Yaskawa INFORM job: A_ROOF_SIDE_0617_2_PAINT_30.JBI

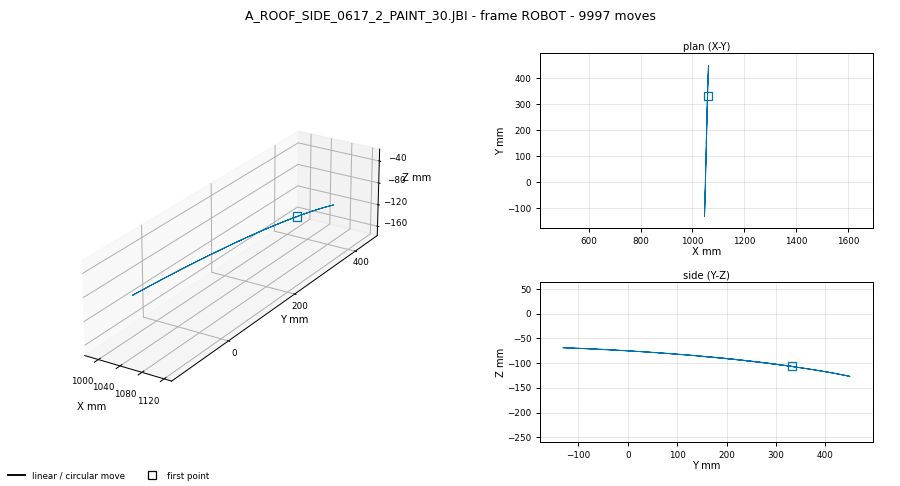
[picture p0: tool path of A_ROOF_SIDE_0617_2_PAINT_30.JBI in frame ROBOT, 9997 of 9997 moves have a stored position in this frame; points joined in program order, loops and branches not executed]
/JOB
//NAME A_ROOF_SIDE_0617_2_PAINT30
//POS
///NPOS 9997,0,0,0,0,0
///TOOL 1
///USER 0
///POSTYPE ROBOT
///RECTAN
///RCONF 1,0,0,0,0,0,0,0,0,0,0,0,0,0,0,0,0,0,0,0,0,0,0,0
C00000=1058.571,332.665,-106.204,173.587,36.326,156.830
C00001=1058.564,332.417,-106.170,173.583,36.321,156.829
C00002=1058.557,332.167,-106.134,173.579,36.317,156.828
C00003=1058.551,331.916,-106.099,173.576,36.312,156.827
C00004=1058.545,331.666,-106.063,173.572,36.307,156.826
C00005=1058.538,331.416,-106.028,173.567,36.303,156.825
C00006=1058.532,331.169,-105.993,173.564,36.298,156.824
C00007=1058.525,330.921,-105.958,173.560,36.294,156.823
C00008=1058.518,330.674,-105.923,173.557,36.289,156.822
C00009=1058.512,330.426,-105.889,173.553,36.285,156.821
C00010=1058.504,330.179,-105.854,173.548,36.280,156.820
C00011=1058.498,329.932,-105.819,173.545,36.276,156.819
C00012=1058.491,329.684,-105.785,173.541,36.271,156.818
C00013=1058.484,329.436,-105.750,173.538,36.267,156.817
C00014=1058.477,329.189,-105.716,173.534,36.262,156.816
C00015=1058.471,328.941,-105.681,173.530,36.258,156.815
C00016=1058.464,328.693,-105.646,173.526,36.254,156.814
C00017=1058.457,328.446,-105.612,173.523,36.249,156.813
C00018=1058.451,328.199,-105.578,173.519,36.245,156.812
C00019=1058.444,327.951,-105.543,173.516,36.241,156.811
C00020=1058.437,327.704,-105.509,173.511,36.237,156.810
C00021=1058.430,327.456,-105.474,173.507,36.232,156.809
C00022=1058.423,327.208,-105.440,173.504,36.227,156.808
C00023=1058.416,326.961,-105.405,173.500,36.223,156.807
C00024=1058.410,326.713,-105.371,173.497,36.219,156.806
C00025=1058.403,326.466,-105.337,173.493,36.215,156.805
C00026=1058.396,326.219,-105.302,173.490,36.210,156.804
C00027=1058.390,325.971,-105.268,173.485,36.206,156.803
C00028=1058.383,325.723,-105.234,173.482,36.202,156.802
C00029=1058.376,325.475,-105.200,173.478,36.197,156.801
C00030=1058.370,325.228,-105.165,173.475,36.193,156.801
C00031=1058.363,324.981,-105.131,173.471,36.189,156.800
C00032=1058.356,324.733,-105.097,173.468,36.184,156.799
C00033=1058.349,324.485,-105.063,173.464,36.180,156.798
C00034=1058.343,324.238,-105.029,173.461,36.176,156.797
C00035=1058.337,323.990,-104.994,173.456,36.171,156.796
C00036=1058.329,323.743,-104.960,173.453,36.167,156.795
C00037=1058.324,323.495,-104.926,173.449,36.163,156.794
C00038=1058.316,323.248,-104.892,173.446,36.159,156.793
C00039=1058.310,323.000,-104.857,173.442,36.154,156.792
C00040=1058.303,322.753,-104.824,173.438,36.150,156.791
C00041=1058.297,322.505,-104.790,173.435,36.145,156.790
C00042=1058.290,322.257,-104.755,173.431,36.141,156.789
C00043=1058.284,322.010,-104.722,173.428,36.137,156.788
C00044=1058.277,321.762,-104.687,173.424,36.133,156.787
C00045=1058.270,321.514,-104.653,173.421,36.128,156.786
C00046=1058.264,321.267,-104.619,173.417,36.124,156.785
C00047=1058.257,321.019,-104.586,173.414,36.120,156.784
C00048=1058.251,320.772,-104.551,173.410,36.116,156.783
C00049=1058.245,320.524,-104.517,173.407,36.112,156.783
C00050=1058.238,320.276,-104.484,173.403,36.107,156.781
C00051=1058.232,320.028,-104.450,173.399,36.103,156.781
C00052=1058.225,319.781,-104.416,173.395,36.099,156.780
C00053=1058.219,319.533,-104.382,173.392,36.094,156.779
C00054=1058.212,319.286,-104.348,173.388,36.090,156.778
C00055=1058.206,319.038,-104.314,173.385,36.086,156.777
C00056=1058.199,318.791,-104.280,173.381,36.082,156.776
C00057=1058.193,318.543,-104.247,173.378,36.078,156.775
C00058=1058.186,318.287,-104.212,173.374,36.073,156.774
C00059=1058.179,318.031,-104.177,173.371,36.069,156.773
C00060=1058.173,317.776,-104.143,173.367,36.064,156.772
C00061=1058.166,317.521,-104.107,173.364,36.060,156.771
C00062=1058.160,317.273,-104.074,173.360,36.056,156.770
C00063=1058.153,317.025,-104.040,173.357,36.052,156.769
C00064=1058.147,316.778,-104.006,173.353,36.047,156.768
C00065=1058.141,316.529,-103.973,173.350,36.043,156.767
C00066=1058.134,316.282,-103.939,173.346,36.039,156.767
C00067=1058.128,316.035,-103.905,173.343,36.034,156.766
C00068=1058.121,315.787,-103.872,173.339,36.030,156.765
C00069=1058.115,315.540,-103.838,173.336,36.026,156.764
C00070=1058.108,315.291,-103.805,173.333,36.022,156.763
C00071=1058.103,315.044,-103.771,173.329,36.018,156.762
C00072=1058.096,314.796,-103.738,173.326,36.014,156.761
C00073=1058.090,314.548,-103.704,173.323,36.010,156.760
C00074=1058.084,314.301,-103.671,173.320,36.006,156.759
C00075=1058.078,314.054,-103.637,173.316,36.001,156.758
C00076=1058.071,313.805,-103.604,173.313,35.997,156.757
C00077=1058.064,313.558,-103.570,173.309,35.993,156.756
C00078=1058.058,313.311,-103.538,173.306,35.989,156.756
C00079=1058.051,313.063,-103.504,173.302,35.985,156.755
C00080=1058.044,312.815,-103.471,173.299,35.981,156.754
C00081=1058.038,312.567,-103.438,173.295,35.977,156.753
C00082=1058.031,312.320,-103.405,173.292,35.973,156.752
C00083=1058.025,312.073,-103.372,173.288,35.969,156.751
C00084=1058.018,311.824,-103.339,173.285,35.964,156.750
C00085=1058.011,311.577,-103.306,173.282,35.960,156.749
C00086=1058.005,311.328,-103.273,173.278,35.956,156.748
C00087=1057.998,311.081,-103.239,173.275,35.952,156.748
C00088=1057.992,310.834,-103.207,173.271,35.948,156.747
C00089=1057.985,310.586,-103.174,173.268,35.944,156.746
C00090=1057.978,310.338,-103.141,173.264,35.940,156.745
C00091=1057.972,310.090,-103.108,173.262,35.937,156.744
C00092=1057.965,309.843,-103.074,173.258,35.933,156.743
C00093=1057.958,309.595,-103.042,173.255,35.929,156.742
C00094=1057.952,309.348,-103.009,173.252,35.924,156.742
C00095=1057.945,309.100,-102.977,173.248,35.920,156.741
C00096=1057.938,308.852,-102.943,173.245,35.916,156.740
C00097=1057.932,308.604,-102.911,173.241,35.912,156.739
C00098=1057.926,308.357,-102.878,173.238,35.908,156.738
C00099=1057.920,308.109,-102.845,173.234,35.904,156.737
C00100=1057.913,307.861,-102.812,173.231,35.901,156.736
C00101=1057.906,307.613,-102.779,173.228,35.897,156.736
C00102=1057.900,307.366,-102.747,173.225,35.893,156.735
C00103=1057.893,307.118,-102.714,173.222,35.888,156.734
C00104=1057.886,306.870,-102.681,173.218,35.884,156.733
C00105=1057.880,306.622,-102.649,173.215,35.880,156.732
C00106=1057.874,306.375,-102.616,173.211,35.876,156.731
C00107=1057.867,306.127,-102.583,173.208,35.873,156.730
C00108=1057.861,305.880,-102.550,173.204,35.869,156.730
C00109=1057.855,305.632,-102.518,173.202,35.865,156.729
C00110=1057.847,305.384,-102.486,173.199,35.861,156.728
C00111=1057.841,305.136,-102.453,173.195,35.857,156.727
C00112=1057.835,304.888,-102.420,173.192,35.852,156.726
C00113=1057.829,304.641,-102.388,173.188,35.849,156.725
C00114=1057.822,304.389,-102.355,173.185,35.845,156.724
C00115=1057.816,304.138,-102.321,173.182,35.841,156.724
C00116=1057.809,303.886,-102.289,173.179,35.837,156.723
C00117=1057.803,303.635,-102.256,173.176,35.833,156.722
C00118=1057.796,303.387,-102.223,173.172,35.829,156.721
C00119=1057.790,303.139,-102.190,173.169,35.825,156.720
C00120=1057.784,302.891,-102.158,173.165,35.820,156.719
C00121=1057.777,302.644,-102.126,173.163,35.817,156.718
C00122=1057.771,302.396,-102.093,173.160,35.813,156.718
C00123=1057.765,302.148,-102.061,173.156,35.809,156.717
C00124=1057.758,301.901,-102.029,173.153,35.805,156.716
C00125=1057.752,301.653,-101.996,173.149,35.801,156.715
C00126=1057.745,301.404,-101.964,173.147,35.797,156.714
C00127=1057.739,301.157,-101.931,173.143,35.793,156.713
C00128=1057.733,300.909,-101.900,173.140,35.789,156.712
C00129=1057.727,300.662,-101.867,173.137,35.785,156.712
C00130=1057.721,300.414,-101.834,173.134,35.781,156.711
C00131=1057.714,300.166,-101.803,173.131,35.777,156.710
C00132=1057.708,299.919,-101.770,173.127,35.773,156.709
C00133=1057.702,299.670,-101.738,173.124,35.769,156.708
C00134=1057.695,299.423,-101.705,173.122,35.766,156.707
C00135=1057.689,299.175,-101.673,173.118,35.762,156.707
C00136=1057.682,298.927,-101.641,173.115,35.757,156.706
C00137=1057.676,298.679,-101.609,173.111,35.753,156.705
C00138=1057.670,298.431,-101.576,173.109,35.750,156.704
C00139=1057.664,298.183,-101.544,173.106,35.746,156.703
C00140=1057.657,297.935,-101.513,173.102,35.742,156.702
C00141=1057.651,297.688,-101.480,173.099,35.738,156.701
C00142=1057.645,297.440,-101.448,173.096,35.734,156.701
C00143=1057.640,297.192,-101.416,173.093,35.730,156.700
C00144=1057.633,296.945,-101.384,173.090,35.726,156.699
C00145=1057.627,296.697,-101.352,173.087,35.722,156.698
C00146=1057.621,296.448,-101.320,173.084,35.718,156.697
C00147=1057.614,296.201,-101.288,173.080,35.714,156.696
C00148=1057.608,295.953,-101.256,173.077,35.711,156.696
C00149=1057.601,295.705,-101.225,173.075,35.707,156.695
C00150=1057.594,295.457,-101.193,173.071,35.703,156.694
C00151=1057.588,295.209,-101.160,173.068,35.699,156.693
C00152=1057.582,294.962,-101.129,173.065,35.695,156.692
C00153=1057.576,294.714,-101.097,173.062,35.691,156.692
C00154=1057.569,294.466,-101.066,173.059,35.687,156.691
C00155=1057.563,294.218,-101.034,173.055,35.684,156.690
C00156=1057.556,293.970,-101.002,173.053,35.680,156.689
C00157=1057.550,293.722,-100.971,173.050,35.676,156.688
C00158=1057.544,293.474,-100.939,173.046,35.672,156.688
C00159=1057.537,293.226,-100.907,173.044,35.669,156.687
C00160=1057.530,292.979,-100.876,173.040,35.664,156.686
C00161=1057.524,292.731,-100.844,173.037,35.661,156.685
C00162=1057.518,292.483,-100.812,173.035,35.657,156.684
C00163=1057.511,292.235,-100.781,173.031,35.653,156.684
C00164=1057.505,291.987,-100.749,173.028,35.649,156.683
C00165=1057.498,291.739,-100.717,173.026,35.646,156.682
C00166=1057.492,291.497,-100.687,173.022,35.642,156.681
C00167=1057.486,291.256,-100.656,173.019,35.638,156.680
C00168=1057.480,291.014,-100.626,173.016,35.635,156.680
C00169=1057.474,290.772,-100.595,173.013,35.630,156.679
C00170=1057.468,290.530,-100.564,173.011,35.627,156.678
C00171=1057.462,290.287,-100.533,173.007,35.623,156.677
C00172=1057.456,290.045,-100.503,173.005,35.620,156.676
C00173=1057.449,289.804,-100.472,173.002,35.616,156.676
C00174=1057.443,289.556,-100.441,172.998,35.612,156.675
C00175=1057.437,289.308,-100.409,172.996,35.608,156.674
C00176=1057.430,289.061,-100.378,172.993,35.605,156.673
C00177=1057.424,288.812,-100.347,172.989,35.601,156.673
C00178=1057.418,288.565,-100.316,172.987,35.597,156.672
C00179=1057.411,288.317,-100.284,172.983,35.593,156.671
C00180=1057.405,288.069,-100.253,172.981,35.589,156.670
C00181=1057.398,287.820,-100.222,172.978,35.586,156.669
C00182=1057.392,287.573,-100.191,172.974,35.582,156.669
C00183=1057.385,287.325,-100.160,172.972,35.578,156.668
C00184=1057.379,287.077,-100.129,172.969,35.575,156.667
C00185=1057.372,286.829,-100.097,172.966,35.571,156.666
C00186=1057.366,286.581,-100.066,172.963,35.567,156.665
C00187=1057.360,286.333,-100.035,172.960,35.563,156.665
C00188=1057.354,286.085,-100.004,172.957,35.560,156.664
C00189=1057.347,285.837,-99.972,172.954,35.556,156.663
C00190=1057.341,285.589,-99.942,172.952,35.552,156.662
C00191=1057.334,285.341,-99.910,172.948,35.549,156.662
C00192=1057.328,285.093,-99.880,172.945,35.545,156.661
C00193=1057.322,284.845,-99.849,172.943,35.541,156.660
C00194=1057.315,284.597,-99.818,172.939,35.538,156.659
C00195=1057.309,284.349,-99.786,172.937,35.533,156.658
C00196=1057.303,284.101,-99.756,172.933,35.530,156.658
C00197=1057.296,283.853,-99.725,172.930,35.526,156.657
C00198=1057.290,283.605,-99.694,172.928,35.522,156.656
C00199=1057.284,283.358,-99.663,172.924,35.519,156.655
C00200=1057.277,283.109,-99.632,172.922,35.515,156.655
C00201=1057.271,282.861,-99.602,172.919,35.511,156.654
C00202=1057.265,282.613,-99.570,172.916,35.508,156.653
C00203=1057.259,282.365,-99.540,172.913,35.504,156.652
C00204=1057.252,282.118,-99.509,172.911,35.500,156.651
C00205=1057.246,281.869,-99.478,172.907,35.496,156.651
C00206=1057.240,281.621,-99.448,172.905,35.493,156.650
C00207=1057.233,281.373,-99.416,172.902,35.489,156.649
C00208=1057.227,281.125,-99.386,172.898,35.485,156.648
C00209=1057.221,280.877,-99.355,172.896,35.482,156.648
C00210=1057.215,280.630,-99.324,172.893,35.477,156.647
C00211=1057.208,280.381,-99.293,172.890,35.474,156.646
C00212=1057.203,280.133,-99.263,172.887,35.470,156.645
C00213=1057.196,279.885,-99.232,172.885,35.466,156.644
C00214=1057.189,279.637,-99.201,172.881,35.463,156.644
C00215=1057.183,279.389,-99.171,172.879,35.459,156.643
C00216=1057.176,279.141,-99.140,172.876,35.456,156.642
C00217=1057.171,278.893,-99.110,172.873,35.451,156.641
C00218=1057.164,278.645,-99.079,172.870,35.448,156.641
C00219=1057.157,278.398,-99.049,172.868,35.444,156.640
C00220=1057.151,278.149,-99.018,172.864,35.441,156.639
C00221=1057.145,277.901,-98.988,172.862,35.437,156.638
C00222=1057.139,277.665,-98.959,172.859,35.434,156.638
C00223=1057.133,277.428,-98.930,172.856,35.430,156.637
C00224=1057.126,277.192,-98.901,172.854,35.427,156.636
C00225=1057.121,276.956,-98.872,172.851,35.423,156.635
C00226=1057.115,276.719,-98.843,172.848,35.420,156.635
C00227=1057.109,276.482,-98.814,172.846,35.416,156.634
C00228=1057.103,276.246,-98.785,172.843,35.412,156.633
C00229=1057.097,276.010,-98.755,172.841,35.409,156.632
C00230=1057.090,275.762,-98.725,172.837,35.405,156.632
C00231=1057.084,275.514,-98.695,172.835,35.402,156.631
C00232=1057.078,275.265,-98.665,172.832,35.398,156.630
C00233=1057.072,275.017,-98.635,172.829,35.394,156.629
C00234=1057.065,274.769,-98.605,172.827,35.391,156.629
C00235=1057.059,274.521,-98.574,172.824,35.387,156.628
C00236=1057.052,274.273,-98.544,172.821,35.383,156.627
C00237=1057.046,274.025,-98.514,172.818,35.379,156.626
C00238=1057.041,273.777,-98.483,172.816,35.376,156.626
C00239=1057.033,273.529,-98.453,172.812,35.372,156.625
C00240=1057.028,273.281,-98.423,172.810,35.369,156.624
C00241=1057.022,273.032,-98.393,172.807,35.365,156.623
C00242=1057.015,272.784,-98.363,172.804,35.361,156.623
C00243=1057.009,272.537,-98.333,172.802,35.357,156.622
C00244=1057.002,272.288,-98.303,172.799,35.354,156.621
C00245=1056.996,272.041,-98.272,172.796,35.350,156.620
C00246=1056.989,271.792,-98.243,172.793,35.347,156.620
C00247=1056.984,271.544,-98.213,172.791,35.343,156.619
C00248=1056.977,271.296,-98.183,172.787,35.339,156.618
C00249=1056.971,271.048,-98.152,172.785,35.335,156.617
C00250=1056.964,270.800,-98.123,172.783,35.332,156.617
C00251=1056.958,270.552,-98.093,172.780,35.328,156.616
C00252=1056.951,270.304,-98.063,172.777,35.325,156.615
C00253=1056.946,270.055,-98.033,172.774,35.321,156.614
C00254=1056.939,269.808,-98.003,172.772,35.318,156.614
C00255=1056.933,269.559,-97.973,172.769,35.314,156.613
C00256=1056.927,269.311,-97.943,172.766,35.310,156.612
C00257=1056.921,269.063,-97.913,172.764,35.306,156.611
C00258=1056.914,268.814,-97.884,172.760,35.303,156.611
C00259=1056.908,268.567,-97.853,172.758,35.299,156.610
C00260=1056.902,268.318,-97.824,172.756,35.296,156.609
C00261=1056.895,268.070,-97.794,172.752,35.292,156.608
C00262=1056.889,267.822,-97.764,172.750,35.289,156.608
C00263=1056.883,267.574,-97.735,172.747,35.285,156.607
C00264=1056.877,267.325,-97.705,172.745,35.281,156.606
C00265=1056.870,267.078,-97.675,172.742,35.277,156.605
C00266=1056.864,266.829,-97.646,172.739,35.274,156.605
C00267=1056.857,266.581,-97.615,172.737,35.270,156.604
C00268=1056.851,266.333,-97.586,172.734,35.267,156.603
C00269=1056.844,266.085,-97.556,172.731,35.263,156.602
C00270=1056.839,265.837,-97.527,172.729,35.259,156.602
C00271=1056.832,265.588,-97.497,172.726,35.256,156.601
C00272=1056.826,265.341,-97.468,172.723,35.252,156.600
C00273=1056.820,265.092,-97.438,172.721,35.249,156.600
C00274=1056.813,264.845,-97.408,172.718,35.245,156.599
C00275=1056.807,264.596,-97.379,172.715,35.241,156.598
C00276=1056.800,264.348,-97.350,172.713,35.237,156.597
C00277=1056.795,264.100,-97.319,172.710,35.234,156.597
C00278=1056.788,263.865,-97.292,172.707,35.230,156.596
C00279=1056.783,263.631,-97.264,172.705,35.227,156.595
C00280=1056.777,263.396,-97.236,172.703,35.224,156.594
C00281=1056.771,263.162,-97.209,172.701,35.220,156.594
C00282=1056.765,262.928,-97.180,172.697,35.217,156.593
C00283=1056.759,262.693,-97.153,172.695,35.214,156.592
C00284=1056.753,262.459,-97.125,172.693,35.210,156.592
C00285=1056.747,262.224,-97.098,172.691,35.206,156.591
C00286=1056.741,261.976,-97.069,172.687,35.203,156.590
C00287=1056.734,261.727,-97.039,172.685,35.200,156.590
C00288=1056.727,261.479,-97.010,172.683,35.196,156.589
C00289=1056.721,261.231,-96.981,172.679,35.193,156.588
C00290=1056.715,260.983,-96.952,172.677,35.189,156.587
C00291=1056.708,260.734,-96.922,172.675,35.186,156.587
C00292=1056.702,260.486,-96.893,172.673,35.182,156.586
C00293=1056.696,260.238,-96.864,172.669,35.178,156.585
C00294=1056.689,259.990,-96.836,172.667,35.175,156.585
C00295=1056.682,259.742,-96.807,172.665,35.171,156.584
C00296=1056.675,259.493,-96.777,172.661,35.168,156.583
C00297=1056.669,259.245,-96.748,172.659,35.164,156.582
C00298=1056.663,258.997,-96.719,172.657,35.161,156.582
C00299=1056.657,258.749,-96.690,172.654,35.157,156.581
C00300=1056.650,258.501,-96.661,172.651,35.153,156.580
C00301=1056.644,258.253,-96.632,172.649,35.150,156.579
C00302=1056.638,258.004,-96.603,172.647,35.146,156.579
C00303=1056.631,257.756,-96.574,172.643,35.143,156.578
C00304=1056.625,257.507,-96.544,172.641,35.139,156.577
C00305=1056.619,257.259,-96.515,172.639,35.135,156.577
C00306=1056.612,257.011,-96.486,172.636,35.132,156.576
C00307=1056.606,256.763,-96.457,172.633,35.128,156.575
C00308=1056.600,256.514,-96.429,172.631,35.125,156.574
C00309=1056.594,256.266,-96.400,172.629,35.121,156.574
C00310=1056.587,256.018,-96.372,172.626,35.118,156.573
C00311=1056.581,255.770,-96.342,172.623,35.114,156.572
C00312=1056.574,255.522,-96.313,172.621,35.110,156.571
C00313=1056.568,255.274,-96.284,172.619,35.107,156.571
C00314=1056.562,255.025,-96.256,172.615,35.103,156.570
C00315=1056.555,254.776,-96.227,172.613,35.100,156.569
C00316=1056.549,254.528,-96.198,172.611,35.096,156.569
C00317=1056.543,254.280,-96.169,172.609,35.092,156.568
C00318=1056.537,254.031,-96.140,172.605,35.089,156.567
C00319=1056.531,253.783,-96.111,172.603,35.085,156.566
C00320=1056.524,253.535,-96.083,172.601,35.082,156.566
C00321=1056.517,253.287,-96.054,172.599,35.078,156.565
C00322=1056.511,253.038,-96.025,172.596,35.075,156.564
C00323=1056.505,252.790,-95.996,172.593,35.070,156.563
C00324=1056.499,252.542,-95.967,172.591,35.067,156.563
C00325=1056.493,252.293,-95.939,172.588,35.063,156.562
C00326=1056.487,252.045,-95.910,172.586,35.060,156.561
C00327=1056.481,251.798,-95.881,172.584,35.056,156.560
C00328=1056.474,251.549,-95.854,172.581,35.052,156.560
C00329=1056.468,251.301,-95.825,172.578,35.049,156.559
C00330=1056.462,251.053,-95.795,172.576,35.045,156.558
C00331=1056.456,250.804,-95.767,172.574,35.042,156.558
C00332=1056.450,250.556,-95.738,172.572,35.038,156.557
C00333=1056.444,250.308,-95.710,172.568,35.034,156.556
C00334=1056.438,250.073,-95.682,172.566,35.031,156.555
C00335=1056.432,249.837,-95.656,172.564,35.027,156.555
C00336=1056.426,249.602,-95.628,172.562,35.024,156.554
C00337=1056.420,249.366,-95.602,172.559,35.021,156.553
C00338=1056.414,249.131,-95.574,172.557,35.017,156.553
C00339=1056.408,248.895,-95.548,172.555,35.014,156.552
C00340=1056.403,248.659,-95.520,172.553,35.010,156.551
C00341=1056.397,248.424,-95.493,172.550,35.007,156.551
C00342=1056.391,248.176,-95.465,172.548,35.003,156.550
C00343=1056.384,247.928,-95.436,172.546,34.999,156.549
C00344=1056.378,247.679,-95.408,172.544,34.996,156.548
C00345=1056.372,247.431,-95.379,172.540,34.992,156.548
C00346=1056.366,247.183,-95.351,172.538,34.988,156.547
C00347=1056.361,246.934,-95.322,172.536,34.985,156.546
C00348=1056.354,246.686,-95.294,172.533,34.981,156.545
C00349=1056.348,246.438,-95.266,172.531,34.978,156.545
C00350=1056.341,246.189,-95.237,172.529,34.973,156.544
C00351=1056.336,245.941,-95.209,172.527,34.970,156.543
C00352=1056.329,245.693,-95.181,172.524,34.966,156.542
C00353=1056.323,245.444,-95.153,172.521,34.963,156.542
C00354=1056.317,245.196,-95.124,172.519,34.959,156.541
C00355=1056.310,244.948,-95.096,172.517,34.955,156.540
C00356=1056.305,244.699,-95.067,172.514,34.952,156.540
C00357=1056.298,244.450,-95.040,172.512,34.948,156.539
C00358=1056.292,244.203,-95.011,172.510,34.945,156.538
C00359=1056.285,243.955,-94.983,172.508,34.941,156.537
C00360=1056.280,243.706,-94.955,172.505,34.937,156.537
C00361=1056.274,243.457,-94.927,172.502,34.934,156.536
C00362=1056.267,243.209,-94.898,172.500,34.930,156.535
C00363=1056.261,242.961,-94.870,172.498,34.927,156.535
C00364=1056.255,242.713,-94.843,172.495,34.923,156.534
C00365=1056.249,242.464,-94.814,172.493,34.919,156.533
C00366=1056.242,242.216,-94.787,172.491,34.916,156.532
C00367=1056.237,241.967,-94.759,172.489,34.912,156.532
C00368=1056.230,241.719,-94.731,172.486,34.909,156.531
C00369=1056.224,241.470,-94.702,172.484,34.905,156.530
C00370=1056.217,241.222,-94.674,172.482,34.901,156.529
C00371=1056.210,240.974,-94.646,172.479,34.898,156.529
C00372=1056.205,240.726,-94.618,172.476,34.894,156.528
C00373=1056.198,240.478,-94.591,172.474,34.891,156.527
C00374=1056.192,240.229,-94.563,172.472,34.887,156.527
C00375=1056.186,239.980,-94.535,172.470,34.883,156.526
C00376=1056.179,239.732,-94.507,172.467,34.880,156.525
C00377=1056.173,239.484,-94.479,172.465,34.876,156.524
C00378=1056.167,239.235,-94.451,172.463,34.873,156.524
C00379=1056.160,238.987,-94.423,172.461,34.869,156.523
C00380=1056.154,238.738,-94.396,172.458,34.865,156.522
C00381=1056.149,238.490,-94.368,172.456,34.862,156.522
C00382=1056.142,238.241,-94.341,172.454,34.858,156.521
C00383=1056.135,237.993,-94.313,172.452,34.855,156.520
C00384=1056.129,237.745,-94.286,172.450,34.851,156.519
C00385=1056.123,237.496,-94.257,172.446,34.847,156.519
C00386=1056.117,237.248,-94.230,172.444,34.844,156.518
C00387=1056.110,237.000,-94.202,172.442,34.840,156.517
C00388=1056.105,236.752,-94.174,172.440,34.837,156.517
C00389=1056.098,236.502,-94.147,172.437,34.832,156.516
C00390=1056.091,236.265,-94.120,172.435,34.829,156.515
C00391=1056.086,236.026,-94.094,172.433,34.826,156.514
C00392=1056.080,235.787,-94.067,172.431,34.822,156.514
C00393=1056.074,235.549,-94.041,172.428,34.818,156.513
C00394=1056.068,235.310,-94.014,172.427,34.815,156.512
C00395=1056.062,235.072,-93.988,172.425,34.812,156.512
C00396=1056.056,234.833,-93.962,172.423,34.808,156.511
C00397=1056.050,234.595,-93.935,172.420,34.805,156.510
C00398=1056.044,234.346,-93.908,172.418,34.801,156.510
C00399=1056.038,234.099,-93.880,172.416,34.797,156.509
C00400=1056.032,233.850,-93.852,172.414,34.794,156.508
C00401=1056.025,233.601,-93.825,172.412,34.790,156.507
C00402=1056.019,233.353,-93.797,172.409,34.787,156.507
C00403=1056.013,233.105,-93.770,172.407,34.783,156.506
C00404=1056.006,232.856,-93.743,172.405,34.779,156.505
C00405=1056.001,232.607,-93.715,172.403,34.775,156.504
C00406=1055.994,232.359,-93.687,172.400,34.772,156.504
C00407=1055.988,232.111,-93.660,172.398,34.768,156.503
C00408=1055.982,231.862,-93.633,172.396,34.764,156.502
C00409=1055.975,231.613,-93.606,172.394,34.761,156.502
C00410=1055.969,231.365,-93.578,172.391,34.757,156.501
C00411=1055.963,231.117,-93.551,172.389,34.754,156.500
C00412=1055.957,230.869,-93.524,172.387,34.750,156.499
C00413=1055.950,230.620,-93.496,172.385,34.746,156.499
C00414=1055.944,230.372,-93.469,172.383,34.743,156.498
C00415=1055.938,230.123,-93.442,172.380,34.739,156.497
C00416=1055.931,229.874,-93.415,172.378,34.735,156.497
C00417=1055.926,229.626,-93.387,172.376,34.732,156.496
C00418=1055.920,229.377,-93.360,172.374,34.728,156.495
C00419=1055.914,229.129,-93.332,172.371,34.724,156.494
C00420=1055.906,228.881,-93.306,172.369,34.720,156.494
C00421=1055.900,228.633,-93.279,172.367,34.717,156.493
C00422=1055.894,228.384,-93.252,172.365,34.713,156.492
C00423=1055.888,228.135,-93.225,172.363,34.710,156.491
C00424=1055.882,227.887,-93.197,172.360,34.706,156.491
C00425=1055.875,227.638,-93.170,172.358,34.702,156.490
C00426=1055.869,227.390,-93.144,172.356,34.699,156.489
C00427=1055.863,227.141,-93.116,172.354,34.695,156.489
C00428=1055.856,226.893,-93.090,172.351,34.691,156.488
C00429=1055.850,226.644,-93.063,172.349,34.688,156.487
C00430=1055.844,226.396,-93.035,172.347,34.684,156.486
C00431=1055.837,226.147,-93.008,172.345,34.681,156.486
C00432=1055.832,225.899,-92.982,172.344,34.677,156.485
C00433=1055.825,225.651,-92.954,172.341,34.673,156.484
C00434=1055.819,225.402,-92.927,172.339,34.670,156.484
C00435=1055.812,225.153,-92.901,172.337,34.666,156.483
C00436=1055.806,224.906,-92.874,172.335,34.663,156.482
C00437=1055.800,224.657,-92.847,172.332,34.659,156.481
C00438=1055.794,224.408,-92.820,172.330,34.655,156.481
C00439=1055.787,224.159,-92.793,172.328,34.651,156.480
C00440=1055.782,223.911,-92.766,172.326,34.647,156.479
C00441=1055.774,223.663,-92.739,172.324,34.644,156.479
C00442=1055.768,223.414,-92.712,172.321,34.640,156.478
C00443=1055.763,223.166,-92.686,172.319,34.637,156.477
C00444=1055.756,222.917,-92.659,172.318,34.633,156.476
C00445=1055.751,222.669,-92.632,172.316,34.629,156.476
C00446=1055.744,222.427,-92.606,172.314,34.626,156.475
C00447=1055.738,222.184,-92.580,172.311,34.622,156.474
C00448=1055.732,221.942,-92.554,172.309,34.618,156.474
C00449=1055.726,221.699,-92.528,172.307,34.615,156.473
C00450=1055.720,221.457,-92.501,172.305,34.611,156.472
C00451=1055.714,221.215,-92.476,172.303,34.608,156.471
C00452=1055.708,220.972,-92.450,172.301,34.604,156.471
C00453=1055.701,220.730,-92.423,172.299,34.600,156.470
C00454=1055.696,220.481,-92.397,172.297,34.597,156.469
C00455=1055.688,220.233,-92.370,172.295,34.593,156.469
C00456=1055.683,219.984,-92.344,172.292,34.589,156.468
C00457=1055.677,219.736,-92.317,172.290,34.586,156.467
C00458=1055.670,219.487,-92.291,172.289,34.582,156.466
C00459=1055.664,219.239,-92.264,172.287,34.578,156.466
C00460=1055.657,218.990,-92.237,172.285,34.574,156.465
C00461=1055.651,218.742,-92.211,172.282,34.571,156.464
C00462=1055.645,218.494,-92.185,172.280,34.567,156.463
C00463=1055.638,218.245,-92.158,172.278,34.564,156.463
C00464=1055.632,217.996,-92.131,172.276,34.560,156.462
C00465=1055.626,217.748,-92.106,172.274,34.556,156.461
C00466=1055.620,217.499,-92.079,172.272,34.553,156.461
C00467=1055.613,217.250,-92.053,172.270,34.549,156.460
C00468=1055.608,217.002,-92.026,172.268,34.545,156.459
C00469=1055.600,216.753,-92.000,172.266,34.541,156.458
C00470=1055.595,216.505,-91.973,172.264,34.538,156.458
C00471=1055.588,216.257,-91.947,172.261,34.534,156.457
C00472=1055.582,216.008,-91.920,172.260,34.530,156.456
C00473=1055.576,215.759,-91.894,172.258,34.527,156.456
C00474=1055.570,215.511,-91.868,172.256,34.523,156.455
C00475=1055.563,215.262,-91.841,172.254,34.519,156.454
C00476=1055.557,215.014,-91.815,172.251,34.515,156.453
C00477=1055.551,214.765,-91.788,172.249,34.512,156.453
C00478=1055.545,214.517,-91.763,172.248,34.508,156.452
C00479=1055.539,214.268,-91.736,172.246,34.504,156.451
C00480=1055.532,214.020,-91.710,172.244,34.501,156.450
C00481=1055.526,213.771,-91.683,172.241,34.496,156.450
C00482=1055.520,213.523,-91.658,172.239,34.493,156.449
C00483=1055.514,213.274,-91.631,172.238,34.489,156.448
C00484=1055.507,213.025,-91.605,172.236,34.486,156.448
C00485=1055.502,212.777,-91.579,172.233,34.481,156.447
C00486=1055.495,212.528,-91.553,172.231,34.478,156.446
C00487=1055.489,212.279,-91.526,172.229,34.474,156.445
C00488=1055.483,212.031,-91.500,172.228,34.470,156.445
C00489=1055.476,211.783,-91.474,172.226,34.467,156.444
C00490=1055.470,211.534,-91.448,172.224,34.463,156.443
C00491=1055.464,211.285,-91.422,172.221,34.459,156.442
C00492=1055.457,211.037,-91.396,172.219,34.455,156.442
C00493=1055.452,210.788,-91.370,172.218,34.452,156.441
C00494=1055.445,210.540,-91.344,172.216,34.448,156.440
C00495=1055.439,210.291,-91.317,172.214,34.444,156.440
C00496=1055.432,210.042,-91.292,172.211,34.440,156.439
C00497=1055.426,209.794,-91.266,172.210,34.437,156.438
C00498=1055.420,209.545,-91.240,172.208,34.433,156.437
C00499=1055.414,209.297,-91.214,172.206,34.429,156.437
C00500=1055.407,209.048,-91.188,172.204,34.426,156.436
C00501=1055.401,208.800,-91.162,172.201,34.421,156.435
C00502=1055.395,208.560,-91.137,172.200,34.418,156.434
C00503=1055.388,208.320,-91.112,172.198,34.414,156.434
C00504=1055.383,208.080,-91.086,172.196,34.411,156.433
C00505=1055.377,207.841,-91.062,172.195,34.407,156.432
C00506=1055.371,207.601,-91.037,172.192,34.403,156.432
C00507=1055.365,207.361,-91.012,172.190,34.400,156.431
C00508=1055.359,207.121,-90.987,172.189,34.396,156.430
C00509=1055.353,206.882,-90.962,172.187,34.393,156.430
C00510=1055.327,205.830,-90.858,171.982,34.302,156.416
C00511=1055.321,205.582,-90.832,171.980,34.299,156.415
C00512=1055.315,205.334,-90.807,171.978,34.296,156.415
C00513=1055.309,205.084,-90.783,171.975,34.293,156.414
C00514=1055.303,204.836,-90.757,171.973,34.290,156.414
C00515=1055.298,204.587,-90.733,171.971,34.287,156.413
C00516=1055.292,204.339,-90.708,171.969,34.284,156.412
C00517=1055.286,204.089,-90.683,171.966,34.281,156.412
C00518=1055.280,203.841,-90.658,171.963,34.278,156.411
C00519=1055.273,203.592,-90.634,171.961,34.276,156.411
C00520=1055.267,203.344,-90.609,171.958,34.272,156.410
C00521=1055.262,203.095,-90.585,171.956,34.269,156.410
C00522=1055.256,202.846,-90.559,171.954,34.267,156.409
C00523=1055.250,202.597,-90.535,171.952,34.264,156.409
C00524=1055.244,202.349,-90.510,171.949,34.261,156.408
C00525=1055.238,202.100,-90.485,171.947,34.258,156.408
C00526=1055.233,201.851,-90.461,171.944,34.255,156.407
C00527=1055.226,201.603,-90.436,171.942,34.252,156.407
C00528=1055.220,201.354,-90.411,171.939,34.249,156.406
C00529=1055.214,201.105,-90.388,171.937,34.246,156.406
C00530=1055.208,200.857,-90.362,171.935,34.244,156.405
C00531=1055.202,200.607,-90.338,171.932,34.241,156.404
C00532=1055.196,200.359,-90.314,171.930,34.238,156.404
C00533=1055.190,200.110,-90.289,171.928,34.235,156.403
C00534=1055.183,199.861,-90.265,171.926,34.233,156.403
C00535=1055.178,199.613,-90.241,171.922,34.229,156.402
C00536=1055.171,199.364,-90.217,171.920,34.227,156.402
C00537=1055.166,199.116,-90.192,171.918,34.224,156.402
C00538=1055.160,198.867,-90.167,171.916,34.221,156.401
C00539=1055.153,198.618,-90.143,171.913,34.219,156.401
C00540=1055.148,198.369,-90.119,171.911,34.216,156.400
C00541=1055.141,198.121,-90.094,171.909,34.213,156.399
C00542=1055.136,197.872,-90.070,171.907,34.210,156.399
C00543=1055.129,197.623,-90.046,171.904,34.207,156.398
C00544=1055.123,197.374,-90.021,171.901,34.204,156.398
C00545=1055.118,197.125,-89.997,171.899,34.202,156.397
C00546=1055.111,196.876,-89.973,171.897,34.199,156.397
C00547=1055.105,196.628,-89.948,171.894,34.196,156.396
C00548=1055.099,196.379,-89.924,171.892,34.194,156.396
C00549=1055.094,196.131,-89.899,171.890,34.191,156.395
C00550=1055.087,195.882,-89.875,171.888,34.188,156.395
C00551=1055.082,195.633,-89.851,171.886,34.185,156.394
C00552=1055.075,195.384,-89.827,171.883,34.182,156.394
C00553=1055.070,195.136,-89.803,171.881,34.179,156.393
C00554=1055.063,194.887,-89.779,171.878,34.177,156.393
C00555=1055.058,194.638,-89.755,171.876,34.174,156.392
C00556=1055.051,194.389,-89.731,171.874,34.171,156.392
C00557=1055.046,194.140,-89.706,171.871,34.169,156.391
C00558=1055.039,193.891,-89.682,171.869,34.166,156.391
C00559=1055.034,193.643,-89.658,171.867,34.163,156.390
C00560=1055.027,193.394,-89.634,171.865,34.160,156.390
C00561=1055.022,193.145,-89.610,171.863,34.157,156.389
C00562=1055.015,192.896,-89.586,171.860,34.155,156.389
C00563=1055.010,192.648,-89.561,171.858,34.152,156.388
C00564=1055.003,192.399,-89.537,171.855,34.149,156.388
C00565=1054.998,192.150,-89.513,171.853,34.146,156.387
C00566=1054.992,191.902,-89.490,171.851,34.144,156.387
C00567=1054.986,191.653,-89.465,171.848,34.141,156.386
C00568=1054.980,191.404,-89.441,171.846,34.138,156.386
C00569=1054.974,191.155,-89.417,171.844,34.135,156.385
C00570=1054.968,190.907,-89.393,171.842,34.133,156.385
C00571=1054.962,190.623,-89.366,171.840,34.130,156.384
C00572=1054.955,190.339,-89.338,171.837,34.126,156.384
C00573=1054.948,190.054,-89.311,171.834,34.123,156.383
C00574=1054.941,189.770,-89.284,171.831,34.120,156.383
C00575=1054.936,189.522,-89.260,171.829,34.117,156.382
C00576=1054.929,189.273,-89.236,171.827,34.115,156.382
C00577=1054.924,189.024,-89.211,171.825,34.112,156.381
C00578=1054.918,188.776,-89.188,171.823,34.109,156.381
C00579=1054.912,188.526,-89.163,171.820,34.106,156.380
C00580=1054.907,188.278,-89.140,171.818,34.103,156.380
C00581=1054.901,188.029,-89.116,171.816,34.101,156.379
C00582=1054.895,187.780,-89.092,171.814,34.098,156.379
C00583=1054.889,187.531,-89.068,171.812,34.095,156.378
C00584=1054.884,187.282,-89.045,171.809,34.093,156.378
C00585=1054.877,187.033,-89.021,171.807,34.090,156.377
C00586=1054.872,186.785,-88.996,171.805,34.087,156.377
C00587=1054.866,186.537,-88.973,171.802,34.084,156.376
C00588=1054.861,186.287,-88.949,171.800,34.081,156.376
C00589=1054.854,186.038,-88.925,171.798,34.079,156.375
C00590=1054.849,185.790,-88.901,171.796,34.076,156.375
C00591=1054.843,185.541,-88.878,171.794,34.073,156.374
C00592=1054.837,185.292,-88.853,171.792,34.071,156.374
C00593=1054.831,185.043,-88.830,171.790,34.068,156.373
C00594=1054.825,184.794,-88.807,171.788,34.065,156.373
C00595=1054.820,184.546,-88.782,171.785,34.063,156.372
C00596=1054.814,184.296,-88.759,171.782,34.059,156.372
C00597=1054.808,184.048,-88.736,171.780,34.057,156.371
C00598=1054.802,183.799,-88.713,171.778,34.054,156.371
C00599=1054.795,183.550,-88.689,171.776,34.052,156.370
C00600=1054.789,183.301,-88.666,171.774,34.049,156.370
C00601=1054.783,183.053,-88.642,171.772,34.047,156.369
C00602=1054.777,182.803,-88.619,171.770,34.044,156.369
C00603=1054.771,182.555,-88.595,171.768,34.042,156.369
C00604=1054.765,182.306,-88.572,171.765,34.039,156.368
C00605=1054.759,182.057,-88.548,171.763,34.037,156.368
C00606=1054.753,181.808,-88.525,171.761,34.034,156.367
C00607=1054.747,181.560,-88.501,171.758,34.032,156.367
C00608=1054.741,181.310,-88.478,171.756,34.029,156.366
C00609=1054.734,181.062,-88.456,171.754,34.027,156.366
C00610=1054.728,180.814,-88.432,171.752,34.024,156.365
C00611=1054.722,180.564,-88.409,171.750,34.021,156.365
C00612=1054.716,180.316,-88.385,171.748,34.018,156.364
C00613=1054.710,180.067,-88.362,171.746,34.016,156.364
C00614=1054.704,179.818,-88.339,171.743,34.013,156.364
C00615=1054.698,179.569,-88.315,171.741,34.011,156.363
C00616=1054.692,179.320,-88.292,171.739,34.008,156.363
C00617=1054.686,179.071,-88.269,171.737,34.006,156.362
C00618=1054.680,178.822,-88.245,171.735,34.003,156.362
C00619=1054.674,178.573,-88.222,171.732,34.001,156.361
C00620=1054.667,178.325,-88.200,171.730,33.998,156.361
C00621=1054.661,178.076,-88.176,171.728,33.996,156.360
C00622=1054.656,177.828,-88.153,171.726,33.993,156.360
C00623=1054.649,177.578,-88.130,171.724,33.991,156.359
C00624=1054.643,177.329,-88.107,171.722,33.988,156.359
C00625=1054.637,177.081,-88.083,171.720,33.985,156.359
C00626=1054.632,176.832,-88.060,171.718,33.983,156.358
C00627=1054.625,176.582,-88.037,171.715,33.980,156.358
C00628=1054.619,176.334,-88.015,171.713,33.978,156.357
C00629=1054.613,176.085,-87.992,171.711,33.975,156.357
C00630=1054.607,175.837,-87.968,171.709,33.973,156.356
C00631=1054.601,175.588,-87.945,171.707,33.970,156.356
C00632=1054.596,175.339,-87.922,171.705,33.968,156.355
C00633=1054.589,175.089,-87.899,171.702,33.965,156.355
C00634=1054.584,174.840,-87.876,171.700,33.963,156.355
C00635=1054.576,174.556,-87.850,171.698,33.959,156.354
C00636=1054.570,174.272,-87.824,171.695,33.956,156.353
C00637=1054.563,173.988,-87.797,171.693,33.954,156.353
C00638=1054.556,173.703,-87.771,171.691,33.951,156.352
C00639=1054.550,173.454,-87.748,171.689,33.948,156.352
C00640=1054.544,173.205,-87.725,171.687,33.946,156.352
C00641=1054.538,172.956,-87.702,171.685,33.943,156.351
C00642=1054.533,172.707,-87.679,171.683,33.941,156.351
C00643=1054.526,172.458,-87.657,171.681,33.938,156.350
C00644=1054.520,172.210,-87.633,171.679,33.935,156.350
C00645=1054.514,171.961,-87.610,171.677,33.933,156.349
C00646=1054.509,171.712,-87.587,171.674,33.930,156.349
C00647=1054.503,171.463,-87.564,171.672,33.928,156.348
C00648=1054.497,171.215,-87.541,171.670,33.925,156.348
C00649=1054.491,170.966,-87.519,171.668,33.923,156.348
C00650=1054.485,170.717,-87.496,171.666,33.920,156.347
C00651=1054.479,170.468,-87.473,171.664,33.918,156.347
C00652=1054.473,170.219,-87.450,171.662,33.915,156.346
C00653=1054.467,169.970,-87.427,171.660,33.913,156.346
C00654=1054.461,169.721,-87.405,171.658,33.910,156.345
C00655=1054.455,169.472,-87.382,171.656,33.908,156.345
C00656=1054.450,169.223,-87.359,171.654,33.905,156.344
C00657=1054.444,168.974,-87.336,171.652,33.902,156.344
C00658=1054.438,168.725,-87.313,171.650,33.900,156.344
C00659=1054.432,168.476,-87.291,171.648,33.897,156.343
C00660=1054.426,168.227,-87.268,171.646,33.895,156.343
C00661=1054.420,167.979,-87.245,171.643,33.892,156.342
C00662=1054.415,167.730,-87.222,171.641,33.890,156.342
C00663=1054.409,167.481,-87.199,171.639,33.887,156.341
C00664=1054.402,167.232,-87.177,171.637,33.885,156.341
C00665=1054.397,166.983,-87.155,171.635,33.882,156.340
C00666=1054.391,166.734,-87.132,171.633,33.880,156.340
C00667=1054.385,166.485,-87.109,171.631,33.877,156.339
C00668=1054.380,166.236,-87.086,171.629,33.875,156.339
C00669=1054.374,165.988,-87.064,171.627,33.872,156.339
C00670=1054.368,165.739,-87.041,171.625,33.870,156.338
C00671=1054.363,165.490,-87.019,171.623,33.866,156.338
C00672=1054.357,165.241,-86.996,171.621,33.864,156.337
C00673=1054.350,164.992,-86.973,171.619,33.861,156.337
C00674=1054.345,164.743,-86.950,171.617,33.859,156.336
C00675=1054.339,164.494,-86.928,171.615,33.856,156.336
C00676=1054.334,164.245,-86.905,171.612,33.854,156.335
C00677=1054.327,163.996,-86.883,171.611,33.851,156.335
C00678=1054.321,163.747,-86.860,171.609,33.849,156.334
C00679=1054.316,163.498,-86.838,171.607,33.846,156.334
C00680=1054.310,163.249,-86.815,171.605,33.844,156.334
C00681=1054.304,163.001,-86.793,171.603,33.841,156.333
C00682=1054.299,162.752,-86.770,171.601,33.838,156.333
C00683=1054.293,162.503,-86.748,171.599,33.836,156.332
C00684=1054.287,162.254,-86.725,171.597,33.833,156.332
C00685=1054.281,162.005,-86.702,171.595,33.831,156.331
C00686=1054.276,161.756,-86.680,171.593,33.828,156.331
C00687=1054.270,161.507,-86.657,171.591,33.826,156.330
C00688=1054.265,161.259,-86.635,171.589,33.823,156.330
C00689=1054.259,161.009,-86.613,171.587,33.821,156.330
C00690=1054.253,160.760,-86.590,171.586,33.818,156.329
C00691=1054.247,160.511,-86.568,171.584,33.816,156.329
C00692=1054.241,160.262,-86.545,171.581,33.814,156.328
C00693=1054.235,160.013,-86.524,171.579,33.811,156.328
C00694=1054.228,159.765,-86.501,171.577,33.809,156.327
C00695=1054.223,159.515,-86.479,171.575,33.806,156.327
C00696=1054.216,159.266,-86.457,171.573,33.804,156.327
C00697=1054.211,159.017,-86.435,171.571,33.801,156.326
C00698=1054.205,158.769,-86.413,171.569,33.799,156.326
C00699=1054.198,158.483,-86.387,171.567,33.796,156.325
C00700=1054.191,158.199,-86.362,171.565,33.793,156.325
C00701=1054.184,157.914,-86.337,171.563,33.790,156.324
C00702=1054.178,157.629,-86.311,171.560,33.788,156.324
C00703=1054.171,157.380,-86.289,171.558,33.785,156.323
C00704=1054.166,157.131,-86.266,171.556,33.782,156.323
C00705=1054.160,156.882,-86.245,171.555,33.781,156.323
C00706=1054.154,156.634,-86.224,171.553,33.778,156.322
C00707=1054.148,156.385,-86.201,171.551,33.776,156.322
C00708=1054.142,156.135,-86.179,171.549,33.773,156.321
C00709=1054.136,155.887,-86.157,171.546,33.770,156.321
C00710=1054.130,155.637,-86.134,171.544,33.768,156.320
C00711=1054.124,155.388,-86.113,171.542,33.766,156.320
C00712=1054.118,155.140,-86.091,171.540,33.763,156.320
C00713=1054.113,154.891,-86.069,171.538,33.761,156.319
C00714=1054.107,154.641,-86.047,171.537,33.758,156.319
C00715=1054.100,154.393,-86.025,171.535,33.756,156.318
C00716=1054.094,154.144,-86.003,171.533,33.754,156.318
C00717=1054.088,153.894,-85.981,171.531,33.751,156.317
C00718=1054.083,153.646,-85.959,171.529,33.749,156.317
C00719=1054.076,153.397,-85.937,171.527,33.747,156.317
C00720=1054.070,153.148,-85.915,171.525,33.744,156.316
C00721=1054.064,152.899,-85.894,171.523,33.742,156.316
C00722=1054.058,152.650,-85.871,171.521,33.739,156.315
C00723=1054.053,152.401,-85.850,171.520,33.737,156.315
C00724=1054.047,152.152,-85.828,171.518,33.735,156.315
C00725=1054.041,151.903,-85.806,171.516,33.732,156.314
C00726=1054.034,151.654,-85.785,171.514,33.730,156.314
C00727=1054.029,151.405,-85.762,171.512,33.727,156.313
C00728=1054.023,151.156,-85.740,171.510,33.725,156.313
C00729=1054.017,150.907,-85.719,171.507,33.723,156.313
C00730=1054.011,150.658,-85.697,171.505,33.720,156.312
C00731=1054.005,150.409,-85.676,171.504,33.717,156.312
C00732=1053.999,150.160,-85.654,171.502,33.716,156.311
C00733=1053.993,149.911,-85.631,171.500,33.713,156.311
C00734=1053.987,149.662,-85.610,171.498,33.710,156.310
C00735=1053.982,149.414,-85.588,171.496,33.708,156.310
C00736=1053.975,149.164,-85.567,171.494,33.706,156.310
C00737=1053.969,148.915,-85.545,171.492,33.703,156.309
C00738=1053.963,148.666,-85.524,171.491,33.701,156.309
C00739=1053.958,148.417,-85.502,171.489,33.698,156.308
C00740=1053.951,148.168,-85.481,171.487,33.696,156.308
C00741=1053.945,147.919,-85.459,171.485,33.694,156.308
C00742=1053.940,147.670,-85.437,171.483,33.691,156.307
C00743=1053.934,147.421,-85.415,171.481,33.689,156.307
C00744=1053.928,147.172,-85.393,171.479,33.687,156.306
C00745=1053.921,146.924,-85.372,171.478,33.684,156.306
C00746=1053.915,146.675,-85.351,171.476,33.682,156.305
C00747=1053.909,146.426,-85.329,171.474,33.680,156.305
C00748=1053.903,146.176,-85.308,171.472,33.677,156.305
C00749=1053.897,145.927,-85.287,171.470,33.675,156.304
C00750=1053.892,145.678,-85.265,171.468,33.673,156.304
C00751=1053.885,145.429,-85.244,171.465,33.670,156.303
C00752=1053.879,145.180,-85.222,171.464,33.668,156.303
C00753=1053.874,144.931,-85.201,171.462,33.666,156.303
C00754=1053.867,144.682,-85.179,171.460,33.663,156.302
C00755=1053.861,144.433,-85.158,171.458,33.661,156.302
C00756=1053.856,144.184,-85.136,171.456,33.659,156.302
C00757=1053.850,143.935,-85.115,171.454,33.656,156.301
C00758=1053.843,143.686,-85.093,171.453,33.654,156.301
C00759=1053.838,143.438,-85.072,171.451,33.652,156.300
C00760=1053.832,143.188,-85.050,171.449,33.649,156.300
C00761=1053.826,142.938,-85.029,171.447,33.646,156.299
C00762=1053.820,142.690,-85.008,171.445,33.644,156.299
C00763=1053.813,142.405,-84.984,171.443,33.641,156.299
C00764=1053.806,142.120,-84.959,171.441,33.639,156.298
C00765=1053.799,141.835,-84.935,171.439,33.636,156.298
C00766=1053.793,141.550,-84.910,171.437,33.634,156.297
C00767=1053.787,141.300,-84.888,171.435,33.631,156.297
C00768=1053.780,141.051,-84.868,171.433,33.628,156.296
C00769=1053.775,140.802,-84.847,171.432,33.627,156.296
C00770=1053.768,140.553,-84.825,171.430,33.624,156.296
C00771=1053.763,140.305,-84.804,171.428,33.621,156.295
C00772=1053.757,140.055,-84.783,171.426,33.620,156.295
C00773=1053.751,139.806,-84.761,171.424,33.617,156.294
C00774=1053.745,139.557,-84.740,171.423,33.614,156.294
C00775=1053.738,139.308,-84.719,171.421,33.613,156.294
C00776=1053.733,139.059,-84.698,171.418,33.610,156.293
C00777=1053.727,138.810,-84.677,171.416,33.608,156.293
C00778=1053.721,138.561,-84.655,171.414,33.605,156.292
C00779=1053.715,138.312,-84.635,171.413,33.603,156.292
C00780=1053.709,138.063,-84.614,171.411,33.601,156.292
C00781=1053.703,137.814,-84.592,171.409,33.598,156.291
C00782=1053.697,137.564,-84.571,171.407,33.596,156.291
C00783=1053.691,137.316,-84.551,171.405,33.594,156.290
C00784=1053.685,137.067,-84.529,171.404,33.591,156.290
C00785=1053.679,136.817,-84.508,171.402,33.589,156.290
C00786=1053.673,136.569,-84.487,171.400,33.587,156.289
C00787=1053.666,136.320,-84.466,171.398,33.584,156.289
C00788=1053.661,136.071,-84.445,171.396,33.582,156.288
C00789=1053.654,135.822,-84.424,171.395,33.580,156.288
C00790=1053.649,135.573,-84.404,171.393,33.578,156.288
C00791=1053.643,135.323,-84.382,171.391,33.575,156.287
C00792=1053.636,135.075,-84.361,171.389,33.573,156.287
C00793=1053.631,134.825,-84.340,171.387,33.571,156.286
C00794=1053.624,134.576,-84.319,171.386,33.568,156.286
C00795=1053.618,134.327,-84.299,171.384,33.566,156.286
C00796=1053.612,134.078,-84.277,171.382,33.564,156.285
C00797=1053.607,133.829,-84.257,171.380,33.561,156.285
C00798=1053.600,133.580,-84.236,171.379,33.559,156.285
C00799=1053.595,133.331,-84.215,171.377,33.557,156.284
C00800=1053.589,133.082,-84.193,171.375,33.555,156.284
C00801=1053.583,132.833,-84.173,171.373,33.552,156.283
C00802=1053.577,132.584,-84.152,171.371,33.550,156.283
C00803=1053.571,132.335,-84.131,171.370,33.548,156.283
C00804=1053.564,132.086,-84.110,171.368,33.545,156.282
C00805=1053.559,131.837,-84.090,171.365,33.543,156.282
C00806=1053.554,131.588,-84.068,171.363,33.541,156.281
C00807=1053.547,131.339,-84.048,171.362,33.538,156.281
C00808=1053.540,131.089,-84.028,171.360,33.536,156.281
C00809=1053.535,130.841,-84.006,171.358,33.534,156.280
C00810=1053.528,130.591,-83.986,171.356,33.532,156.280
C00811=1053.523,130.342,-83.966,171.354,33.529,156.279
C00812=1053.516,130.093,-83.945,171.353,33.527,156.279
C00813=1053.510,129.844,-83.925,171.351,33.525,156.279
C00814=1053.504,129.594,-83.904,171.349,33.523,156.278
C00815=1053.498,129.346,-83.883,171.347,33.521,156.278
C00816=1053.491,129.097,-83.863,171.346,33.518,156.278
C00817=1053.486,128.848,-83.842,171.344,33.516,156.277
C00818=1053.479,128.599,-83.821,171.342,33.514,156.277
C00819=1053.473,128.350,-83.801,171.340,33.512,156.276
C00820=1053.467,128.100,-83.780,171.339,33.509,156.276
C00821=1053.461,127.852,-83.760,171.337,33.507,156.276
C00822=1053.456,127.603,-83.739,171.335,33.505,156.275
C00823=1053.449,127.353,-83.719,171.333,33.503,156.275
C00824=1053.443,127.104,-83.699,171.332,33.500,156.274
C00825=1053.437,126.855,-83.677,171.330,33.498,156.274
C00826=1053.431,126.606,-83.657,171.328,33.495,156.274
C00827=1053.424,126.321,-83.633,171.326,33.493,156.273
C00828=1053.417,126.036,-83.610,171.324,33.490,156.273
C00829=1053.410,125.750,-83.587,171.322,33.488,156.272
C00830=1053.403,125.464,-83.563,171.320,33.485,156.272
C00831=1053.397,125.215,-83.543,171.318,33.483,156.272
C00832=1053.390,124.967,-83.522,171.316,33.481,156.271
C00833=1053.385,124.717,-83.502,171.315,33.479,156.271
C00834=1053.379,124.469,-83.482,171.313,33.476,156.270
C00835=1053.373,124.219,-83.461,171.311,33.474,156.270
C00836=1053.367,123.970,-83.441,171.310,33.472,156.270
C00837=1053.361,123.720,-83.420,171.308,33.470,156.269
C00838=1053.354,123.472,-83.400,171.306,33.467,156.269
C00839=1053.348,123.223,-83.380,171.304,33.465,156.269
C00840=1053.343,122.974,-83.359,171.303,33.463,156.268
C00841=1053.337,122.725,-83.339,171.301,33.460,156.268
C00842=1053.331,122.476,-83.319,171.298,33.458,156.267
C00843=1053.325,122.226,-83.298,171.296,33.455,156.267
C00844=1053.319,121.977,-83.278,171.295,33.454,156.267
C00845=1053.313,121.729,-83.258,171.293,33.451,156.266
C00846=1053.307,121.479,-83.237,171.291,33.449,156.266
C00847=1053.301,121.230,-83.217,171.290,33.447,156.265
C00848=1053.295,120.981,-83.197,171.288,33.445,156.265
C00849=1053.288,120.732,-83.176,171.286,33.442,156.265
C00850=1053.283,120.483,-83.156,171.284,33.440,156.264
C00851=1053.277,120.234,-83.136,171.283,33.438,156.264
C00852=1053.270,119.985,-83.115,171.281,33.436,156.264
C00853=1053.265,119.736,-83.095,171.279,33.433,156.263
C00854=1053.259,119.487,-83.075,171.278,33.431,156.263
C00855=1053.252,119.237,-83.055,171.276,33.428,156.262
C00856=1053.246,118.989,-83.035,171.274,33.426,156.262
C00857=1053.241,118.739,-83.014,171.272,33.424,156.262
C00858=1053.235,118.491,-82.994,171.271,33.421,156.261
C00859=1053.229,118.240,-82.975,171.269,33.419,156.261
C00860=1053.224,117.991,-82.954,171.267,33.417,156.260
C00861=1053.218,117.742,-82.934,171.266,33.415,156.260
C00862=1053.212,117.494,-82.914,171.264,33.412,156.260
C00863=1053.205,117.244,-82.894,171.262,33.410,156.259
C00864=1053.200,116.995,-82.873,171.260,33.408,156.259
C00865=1053.194,116.746,-82.853,171.259,33.405,156.258
C00866=1053.188,116.497,-82.833,171.257,33.403,156.258
C00867=1053.181,116.248,-82.813,171.255,33.401,156.258
C00868=1053.176,115.999,-82.792,171.254,33.399,156.257
C00869=1053.170,115.750,-82.772,171.252,33.396,156.257
C00870=1053.164,115.501,-82.752,171.250,33.394,156.257
C00871=1053.158,115.251,-82.733,171.249,33.392,156.256
C00872=1053.152,115.002,-82.712,171.247,33.389,156.256
C00873=1053.146,114.753,-82.692,171.245,33.387,156.255
C00874=1053.140,114.504,-82.672,171.244,33.385,156.255
C00875=1053.134,114.255,-82.652,171.242,33.383,156.255
C00876=1053.128,114.006,-82.632,171.240,33.380,156.254
C00877=1053.123,113.756,-82.612,171.239,33.378,156.254
C00878=1053.117,113.507,-82.592,171.237,33.376,156.254
C00879=1053.111,113.259,-82.572,171.235,33.374,156.253
C00880=1053.105,113.010,-82.552,171.233,33.371,156.253
C00881=1053.099,112.760,-82.533,171.232,33.369,156.252
C00882=1053.093,112.511,-82.513,171.230,33.367,156.252
C00883=1053.087,112.262,-82.493,171.228,33.365,156.252
C00884=1053.081,112.013,-82.473,171.227,33.362,156.251
C00885=1053.074,111.763,-82.453,171.225,33.360,156.251
C00886=1053.068,111.514,-82.433,171.223,33.357,156.250
C00887=1053.062,111.265,-82.413,171.222,33.356,156.250
C00888=1053.057,111.016,-82.394,171.220,33.354,156.250
C00889=1053.051,110.767,-82.374,171.218,33.351,156.249
C00890=1053.043,110.518,-82.354,171.217,33.349,156.249
C00891=1053.037,110.233,-82.332,171.215,33.346,156.249
C00892=1053.030,109.947,-82.310,171.213,33.344,156.248
C00893=1053.023,109.661,-82.287,171.210,33.341,156.248
C00894=1053.016,109.376,-82.265,171.208,33.339,156.247
C00895=1053.010,109.127,-82.245,171.206,33.337,156.247
C00896=1053.004,108.878,-82.224,171.204,33.334,156.247
C00897=1052.998,108.628,-82.205,171.203,33.332,156.246
C00898=1052.991,108.380,-82.186,171.201,33.330,156.246
C00899=1052.985,108.130,-82.166,171.199,33.328,156.246
C00900=1052.979,107.881,-82.147,171.198,33.326,156.245
C00901=1052.973,107.631,-82.127,171.196,33.323,156.245
C00902=1052.967,107.382,-82.107,171.194,33.321,156.244
C00903=1052.961,107.134,-82.087,171.193,33.319,156.244
C00904=1052.955,106.885,-82.068,171.191,33.317,156.244
C00905=1052.949,106.636,-82.048,171.189,33.315,156.243
C00906=1052.943,106.386,-82.029,171.188,33.312,156.243
C00907=1052.937,106.138,-82.009,171.186,33.310,156.243
C00908=1052.931,105.887,-81.990,171.184,33.308,156.242
C00909=1052.925,105.639,-81.970,171.183,33.306,156.242
C00910=1052.918,105.389,-81.951,171.181,33.303,156.241
C00911=1052.912,105.141,-81.931,171.179,33.301,156.241
C00912=1052.907,104.891,-81.912,171.178,33.299,156.241
C00913=1052.901,104.642,-81.892,171.176,33.297,156.240
C00914=1052.895,104.393,-81.873,171.174,33.295,156.240
C00915=1052.888,104.144,-81.853,171.173,33.292,156.240
C00916=1052.882,103.894,-81.834,171.171,33.290,156.239
C00917=1052.876,103.645,-81.814,171.169,33.287,156.239
C00918=1052.870,103.396,-81.794,171.168,33.286,156.239
C00919=1052.865,103.147,-81.775,171.166,33.283,156.238
C00920=1052.858,102.898,-81.756,171.164,33.281,156.238
C00921=1052.852,102.649,-81.737,171.163,33.279,156.237
C00922=1052.847,102.399,-81.717,171.161,33.276,156.237
C00923=1052.841,102.150,-81.697,171.159,33.274,156.237
C00924=1052.835,101.901,-81.678,171.158,33.272,156.236
C00925=1052.828,101.653,-81.659,171.156,33.270,156.236
C00926=1052.822,101.403,-81.639,171.154,33.267,156.236
C00927=1052.817,101.154,-81.620,171.153,33.265,156.235
C00928=1052.811,100.905,-81.600,171.151,33.263,156.235
C00929=1052.805,100.655,-81.581,171.149,33.261,156.234
C00930=1052.798,100.406,-81.562,171.148,33.259,156.234
C00931=1052.792,100.157,-81.542,171.146,33.256,156.234
C00932=1052.786,99.908,-81.523,171.144,33.254,156.233
C00933=1052.780,99.658,-81.504,171.143,33.252,156.233
C00934=1052.773,99.409,-81.486,171.141,33.250,156.233
C00935=1052.767,99.160,-81.466,171.139,33.248,156.232
C00936=1052.761,98.911,-81.447,171.138,33.245,156.232
C00937=1052.755,98.662,-81.428,171.136,33.243,156.232
C00938=1052.750,98.412,-81.408,171.134,33.241,156.231
C00939=1052.743,98.164,-81.389,171.133,33.239,156.231
C00940=1052.737,97.914,-81.370,171.131,33.237,156.230
C00941=1052.731,97.665,-81.351,171.129,33.235,156.230
C00942=1052.725,97.416,-81.332,171.128,33.232,156.230
C00943=1052.719,97.167,-81.313,171.126,33.230,156.229
C00944=1052.713,96.918,-81.293,171.124,33.228,156.229
C00945=1052.706,96.669,-81.275,171.123,33.226,156.229
C00946=1052.701,96.419,-81.255,171.121,33.224,156.228
C00947=1052.695,96.170,-81.236,171.119,33.221,156.228
C00948=1052.689,95.921,-81.218,171.118,33.219,156.228
C00949=1052.683,95.671,-81.198,171.116,33.217,156.227
C00950=1052.676,95.423,-81.179,171.114,33.215,156.227
C00951=1052.670,95.173,-81.160,171.113,33.213,156.226
C00952=1052.664,94.924,-81.141,171.111,33.211,156.226
C00953=1052.658,94.675,-81.122,171.109,33.208,156.226
C00954=1052.652,94.426,-81.103,171.108,33.206,156.225
C00955=1052.644,94.140,-81.081,171.106,33.204,156.225
C00956=1052.638,93.854,-81.060,171.104,33.201,156.225
C00957=1052.631,93.569,-81.038,171.102,33.198,156.224
C00958=1052.624,93.283,-81.016,171.100,33.196,156.224
C00959=1052.618,93.034,-80.997,171.099,33.194,156.223
C00960=1052.612,92.786,-80.978,171.097,33.191,156.223
C00961=1052.606,92.536,-80.958,171.095,33.189,156.223
C00962=1052.600,92.287,-80.940,171.094,33.187,156.222
C00963=1052.594,92.038,-80.921,171.092,33.185,156.222
C00964=1052.588,91.789,-80.902,171.090,33.183,156.222
C00965=1052.582,91.539,-80.883,171.089,33.180,156.221
C00966=1052.576,91.290,-80.864,171.087,33.178,156.221
C00967=1052.570,91.041,-80.845,171.086,33.176,156.220
C00968=1052.564,90.792,-80.826,171.084,33.174,156.220
C00969=1052.558,90.542,-80.807,171.082,33.172,156.220
C00970=1052.552,90.293,-80.788,171.081,33.169,156.219
C00971=1052.545,90.044,-80.770,171.079,33.167,156.219
C00972=1052.539,89.794,-80.752,171.077,33.165,156.219
C00973=1052.533,89.545,-80.732,171.076,33.163,156.218
C00974=1052.527,89.296,-80.714,171.074,33.161,156.218
C00975=1052.520,89.047,-80.695,171.072,33.159,156.218
C00976=1052.514,88.797,-80.676,171.071,33.157,156.217
C00977=1052.509,88.549,-80.658,171.069,33.154,156.217
C00978=1052.502,88.300,-80.639,171.067,33.152,156.217
C00979=1052.496,88.050,-80.620,171.066,33.150,156.216
C00980=1052.490,87.801,-80.602,171.064,33.148,156.216
C00981=1052.484,87.551,-80.583,171.062,33.146,156.215
C00982=1052.478,87.302,-80.564,171.061,33.144,156.215
C00983=1052.471,87.053,-80.546,171.059,33.142,156.215
C00984=1052.465,86.804,-80.527,171.058,33.139,156.214
C00985=1052.459,86.554,-80.508,171.056,33.137,156.214
C00986=1052.453,86.305,-80.489,171.054,33.135,156.214
C00987=1052.447,86.056,-80.471,171.053,33.133,156.213
C00988=1052.441,85.807,-80.453,171.051,33.131,156.213
C00989=1052.435,85.558,-80.434,171.049,33.129,156.213
C00990=1052.429,85.309,-80.415,171.048,33.126,156.212
C00991=1052.422,85.060,-80.397,171.046,33.124,156.212
C00992=1052.416,84.810,-80.379,171.044,33.122,156.212
C00993=1052.410,84.561,-80.360,171.043,33.120,156.211
C00994=1052.404,84.311,-80.341,171.041,33.118,156.211
C00995=1052.398,84.062,-80.322,171.040,33.116,156.211
C00996=1052.392,83.813,-80.304,171.038,33.113,156.210
C00997=1052.386,83.564,-80.286,171.036,33.111,156.210
C00998=1052.379,83.315,-80.267,171.035,33.109,156.210
C00999=1052.374,83.065,-80.248,171.033,33.107,156.209
C01000=1052.368,82.816,-80.230,171.031,33.105,156.209
C01001=1052.361,82.567,-80.211,171.030,33.103,156.208
C01002=1052.355,82.318,-80.193,171.028,33.100,156.208
C01003=1052.349,82.068,-80.175,171.026,33.098,156.208
C01004=1052.343,81.819,-80.156,171.025,33.096,156.207
C01005=1052.337,81.570,-80.137,171.023,33.093,156.207
C01006=1052.331,81.320,-80.119,171.022,33.092,156.207
C01007=1052.325,81.072,-80.101,171.020,33.090,156.206
C01008=1052.319,80.823,-80.082,171.018,33.087,156.206
C01009=1052.313,80.572,-80.064,171.017,33.085,156.206
C01010=1052.307,80.323,-80.045,171.015,33.083,156.205
C01011=1052.301,80.075,-80.027,171.013,33.080,156.205
C01012=1052.295,79.825,-80.009,171.012,33.078,156.205
C01013=1052.289,79.576,-79.990,171.010,33.076,156.204
C01014=1052.282,79.327,-79.972,171.009,33.074,156.204
C01015=1052.277,79.077,-79.953,171.007,33.072,156.203
C01016=1052.271,78.828,-79.935,171.005,33.069,156.203
C01017=1052.265,78.579,-79.917,171.004,33.067,156.203
C01018=1052.258,78.330,-79.898,171.002,33.065,156.202
C01019=1052.251,78.044,-79.878,171.000,33.063,156.202
C01020=1052.245,77.759,-79.856,170.998,33.060,156.202
C01021=1052.237,77.473,-79.836,170.996,33.058,156.201
C01022=1052.231,77.188,-79.814,170.995,33.056,156.201
C01023=1052.224,76.938,-79.797,170.993,33.053,156.200
C01024=1052.217,76.689,-79.778,170.991,33.051,156.200
C01025=1052.211,76.439,-79.761,170.990,33.049,156.200
C01026=1052.205,76.191,-79.742,170.988,33.047,156.199
C01027=1052.199,75.941,-79.724,170.986,33.044,156.199
C01028=1052.193,75.692,-79.706,170.985,33.042,156.199
C01029=1052.187,75.442,-79.688,170.983,33.040,156.198
C01030=1052.181,75.193,-79.670,170.982,33.039,156.198
C01031=1052.175,74.944,-79.652,170.980,33.036,156.198
C01032=1052.169,74.695,-79.634,170.978,33.034,156.197
C01033=1052.162,74.445,-79.615,170.977,33.032,156.197
C01034=1052.157,74.196,-79.597,170.975,33.030,156.197
C01035=1052.150,73.947,-79.579,170.973,33.027,156.196
C01036=1052.144,73.697,-79.561,170.972,33.025,156.196
C01037=1052.139,73.448,-79.543,170.970,33.023,156.196
C01038=1052.132,73.200,-79.525,170.968,33.021,156.195
C01039=1052.125,72.950,-79.507,170.967,33.019,156.195
C01040=1052.119,72.701,-79.489,170.965,33.017,156.195
C01041=1052.114,72.452,-79.471,170.964,33.015,156.194
C01042=1052.107,72.202,-79.453,170.962,33.012,156.194
C01043=1052.101,71.953,-79.434,170.960,33.010,156.193
C01044=1052.095,71.704,-79.417,170.959,33.008,156.193
C01045=1052.089,71.454,-79.399,170.957,33.006,156.193
C01046=1052.083,71.205,-79.380,170.955,33.004,156.192
C01047=1052.077,70.956,-79.363,170.954,33.002,156.192
C01048=1052.071,70.707,-79.345,170.952,33.000,156.192
C01049=1052.064,70.457,-79.327,170.951,32.997,156.191
C01050=1052.059,70.208,-79.309,170.949,32.995,156.191
C01051=1052.052,69.959,-79.291,170.947,32.993,156.191
C01052=1052.046,69.709,-79.273,170.946,32.991,156.190
C01053=1052.041,69.460,-79.255,170.944,32.989,156.190
C01054=1052.034,69.211,-79.238,170.943,32.987,156.190
C01055=1052.028,68.961,-79.220,170.942,32.985,156.189
C01056=1052.022,68.712,-79.202,170.940,32.983,156.189
C01057=1052.016,68.462,-79.184,170.939,32.980,156.189
C01058=1052.009,68.214,-79.166,170.937,32.978,156.188
C01059=1052.003,67.965,-79.149,170.935,32.976,156.188
C01060=1051.997,67.715,-79.131,170.934,32.974,156.188
C01061=1051.991,67.465,-79.113,170.932,32.972,156.187
C01062=1051.985,67.216,-79.096,170.930,32.970,156.187
C01063=1051.978,66.967,-79.077,170.929,32.968,156.187
C01064=1051.973,66.718,-79.060,170.927,32.966,156.186
C01065=1051.967,66.469,-79.042,170.925,32.964,156.186
C01066=1051.960,66.219,-79.024,170.924,32.961,156.186
C01067=1051.954,65.970,-79.007,170.922,32.959,156.185
C01068=1051.948,65.720,-78.989,170.921,32.957,156.185
C01069=1051.941,65.472,-78.971,170.919,32.955,156.185
C01070=1051.935,65.222,-78.953,170.917,32.953,156.184
C01071=1051.929,64.973,-78.935,170.916,32.951,156.184
C01072=1051.923,64.724,-78.918,170.914,32.949,156.184
C01073=1051.917,64.474,-78.900,170.912,32.946,156.183
C01074=1051.911,64.225,-78.882,170.911,32.945,156.183
C01075=1051.905,63.976,-78.865,170.909,32.942,156.183
C01076=1051.898,63.726,-78.847,170.907,32.940,156.182
C01077=1051.892,63.477,-78.831,170.906,32.938,156.182
C01078=1051.886,63.228,-78.813,170.904,32.936,156.182
C01079=1051.879,62.978,-78.795,170.903,32.934,156.181
C01080=1051.874,62.729,-78.778,170.901,32.932,156.181
C01081=1051.867,62.480,-78.760,170.899,32.930,156.181
C01082=1051.860,62.230,-78.743,170.898,32.928,156.180
C01083=1051.853,61.944,-78.723,170.896,32.925,156.180
C01084=1051.846,61.659,-78.702,170.894,32.923,156.180
C01085=1051.839,61.373,-78.682,170.892,32.921,156.179
C01086=1051.831,61.087,-78.663,170.890,32.919,156.179
C01087=1051.826,60.838,-78.646,170.888,32.916,156.178
C01088=1051.819,60.589,-78.628,170.887,32.914,156.178
C01089=1051.813,60.340,-78.611,170.885,32.912,156.178
C01090=1051.806,60.091,-78.593,170.883,32.910,156.178
C01091=1051.801,59.841,-78.576,170.882,32.908,156.177
C01092=1051.794,59.592,-78.558,170.880,32.906,156.177
C01093=1051.787,59.343,-78.541,170.878,32.904,156.177
C01094=1051.782,59.094,-78.523,170.877,32.902,156.176
C01095=1051.775,58.844,-78.507,170.875,32.900,156.176
C01096=1051.770,58.594,-78.489,170.874,32.898,156.176
C01097=1051.763,58.345,-78.472,170.872,32.896,156.175
C01098=1051.756,58.096,-78.455,170.870,32.894,156.175
C01099=1051.750,57.847,-78.437,170.869,32.892,156.175
C01100=1051.744,57.598,-78.420,170.867,32.890,156.174
C01101=1051.738,57.348,-78.402,170.865,32.888,156.174
C01102=1051.731,57.098,-78.386,170.864,32.886,156.174
C01103=1051.725,56.849,-78.369,170.862,32.884,156.173
C01104=1051.719,56.600,-78.351,170.860,32.881,156.173
C01105=1051.713,56.351,-78.334,170.859,32.879,156.173
C01106=1051.707,56.101,-78.316,170.857,32.877,156.172
C01107=1051.700,55.852,-78.299,170.855,32.875,156.172
C01108=1051.694,55.602,-78.282,170.855,32.873,156.172
C01109=1051.688,55.353,-78.265,170.853,32.871,156.171
C01110=1051.681,55.104,-78.247,170.852,32.869,156.171
C01111=1051.676,54.855,-78.230,170.850,32.867,156.171
C01112=1051.670,54.605,-78.213,170.848,32.864,156.170
C01113=1051.663,54.356,-78.196,170.847,32.863,156.170
C01114=1051.658,54.107,-78.178,170.845,32.861,156.170
C01115=1051.651,53.858,-78.161,170.843,32.858,156.169
C01116=1051.645,53.608,-78.145,170.842,32.857,156.169
C01117=1051.639,53.359,-78.127,170.840,32.855,156.169
C01118=1051.632,53.110,-78.110,170.838,32.852,156.168
C01119=1051.626,52.860,-78.092,170.837,32.850,156.168
C01120=1051.620,52.611,-78.076,170.835,32.848,156.168
C01121=1051.613,52.361,-78.058,170.833,32.846,156.167
C01122=1051.608,52.112,-78.041,170.832,32.844,156.167
C01123=1051.602,51.863,-78.025,170.830,32.842,156.167
C01124=1051.595,51.613,-78.007,170.829,32.839,156.166
C01125=1051.590,51.364,-77.990,170.827,32.837,156.166
C01126=1051.583,51.114,-77.973,170.825,32.835,156.166
C01127=1051.577,50.866,-77.956,170.824,32.833,156.165
C01128=1051.571,50.617,-77.939,170.822,32.831,156.165
C01129=1051.565,50.367,-77.922,170.820,32.829,156.165
C01130=1051.558,50.118,-77.905,170.819,32.827,156.164
C01131=1051.553,49.867,-77.888,170.817,32.825,156.164
C01132=1051.546,49.619,-77.871,170.815,32.823,156.164
C01133=1051.540,49.370,-77.854,170.814,32.821,156.163
C01134=1051.534,49.120,-77.837,170.812,32.819,156.163
C01135=1051.528,48.871,-77.820,170.810,32.817,156.163
C01136=1051.522,48.622,-77.803,170.809,32.814,156.162
C01137=1051.516,48.372,-77.785,170.807,32.812,156.162
C01138=1051.510,48.123,-77.768,170.806,32.810,156.162
C01139=1051.503,47.873,-77.752,170.804,32.808,156.161
C01140=1051.498,47.624,-77.734,170.802,32.806,156.161
C01141=1051.492,47.375,-77.718,170.801,32.804,156.161
C01142=1051.485,47.125,-77.701,170.799,32.802,156.160
C01143=1051.480,46.876,-77.684,170.797,32.800,156.160
C01144=1051.473,46.627,-77.667,170.796,32.798,156.160
C01145=1051.467,46.377,-77.650,170.794,32.796,156.160
C01146=1051.461,46.128,-77.633,170.792,32.794,156.159
C01147=1051.454,45.841,-77.614,170.792,32.791,156.159
C01148=1051.448,45.556,-77.594,170.790,32.788,156.158
C01149=1051.441,45.270,-77.575,170.788,32.786,156.158
C01150=1051.433,44.984,-77.556,170.786,32.784,156.158
C01151=1051.428,44.734,-77.539,170.784,32.782,156.157
C01152=1051.421,44.485,-77.522,170.783,32.780,156.157
C01153=1051.415,44.236,-77.505,170.781,32.777,156.157
C01154=1051.410,43.987,-77.488,170.779,32.775,156.156
C01155=1051.404,43.737,-77.472,170.778,32.773,156.156
C01156=1051.397,43.488,-77.454,170.776,32.771,156.156
C01157=1051.391,43.238,-77.438,170.774,32.769,156.155
C01158=1051.385,42.989,-77.422,170.773,32.767,156.155
C01159=1051.378,42.740,-77.404,170.771,32.765,156.155
C01160=1051.372,42.490,-77.388,170.769,32.763,156.154
C01161=1051.366,42.241,-77.372,170.768,32.760,156.154
C01162=1051.360,41.991,-77.354,170.766,32.758,156.154
C01163=1051.354,41.742,-77.338,170.764,32.756,156.153
C01164=1051.348,41.493,-77.321,170.763,32.754,156.153
C01165=1051.341,41.243,-77.304,170.761,32.752,156.153
C01166=1051.335,40.994,-77.288,170.759,32.750,156.152
C01167=1051.329,40.744,-77.272,170.758,32.748,156.152
C01168=1051.323,40.496,-77.255,170.756,32.746,156.152
C01169=1051.317,40.246,-77.238,170.754,32.744,156.152
C01170=1051.311,39.996,-77.222,170.753,32.742,156.151
C01171=1051.304,39.748,-77.205,170.751,32.740,156.151
C01172=1051.298,39.498,-77.188,170.749,32.738,156.151
C01173=1051.292,39.248,-77.172,170.748,32.736,156.150
C01174=1051.286,38.999,-77.156,170.746,32.734,156.150
C01175=1051.280,38.750,-77.139,170.744,32.732,156.150
C01176=1051.274,38.501,-77.122,170.743,32.730,156.149
C01177=1051.267,38.251,-77.106,170.741,32.728,156.149
C01178=1051.261,38.001,-77.089,170.740,32.726,156.149
C01179=1051.255,37.753,-77.073,170.739,32.724,156.148
C01180=1051.249,37.503,-77.056,170.737,32.722,156.148
C01181=1051.242,37.253,-77.040,170.735,32.720,156.148
C01182=1051.237,37.004,-77.023,170.734,32.718,156.147
C01183=1051.231,36.755,-77.007,170.732,32.716,156.147
C01184=1051.225,36.505,-76.991,170.730,32.714,156.147
C01185=1051.218,36.256,-76.974,170.729,32.712,156.146
C01186=1051.211,36.007,-76.958,170.727,32.710,156.146
C01187=1051.205,35.757,-76.942,170.725,32.708,156.146
C01188=1051.199,35.508,-76.925,170.724,32.706,156.146
C01189=1051.193,35.258,-76.909,170.722,32.704,156.145
C01190=1051.187,35.009,-76.892,170.720,32.701,156.145
C01191=1051.181,34.759,-76.876,170.719,32.700,156.145
C01192=1051.174,34.510,-76.861,170.717,32.698,156.144
C01193=1051.168,34.261,-76.844,170.715,32.695,156.144
C01194=1051.161,34.011,-76.827,170.714,32.694,156.144
C01195=1051.155,33.762,-76.811,170.712,32.691,156.143
C01196=1051.149,33.513,-76.794,170.710,32.689,156.143
C01197=1051.143,33.264,-76.779,170.709,32.687,156.143
C01198=1051.137,33.014,-76.763,170.707,32.685,156.143
C01199=1051.130,32.764,-76.746,170.705,32.683,156.142
C01200=1051.124,32.515,-76.730,170.704,32.681,156.142
C01201=1051.118,32.266,-76.713,170.702,32.679,156.142
C01202=1051.112,32.016,-76.697,170.700,32.677,156.141
C01203=1051.106,31.767,-76.681,170.698,32.675,156.141
C01204=1051.100,31.518,-76.665,170.697,32.674,156.141
C01205=1051.093,31.268,-76.649,170.695,32.672,156.140
C01206=1051.087,31.018,-76.632,170.694,32.670,156.140
C01207=1051.081,30.769,-76.616,170.693,32.668,156.140
C01208=1051.074,30.520,-76.600,170.691,32.666,156.140
C01209=1051.069,30.271,-76.584,170.689,32.664,156.139
C01210=1051.063,30.021,-76.568,170.688,32.662,156.139
C01211=1051.055,29.735,-76.549,170.686,32.659,156.139
C01212=1051.048,29.450,-76.531,170.684,32.657,156.138
C01213=1051.041,29.163,-76.512,170.682,32.655,156.138
C01214=1051.034,28.877,-76.494,170.680,32.652,156.138
C01215=1051.028,28.627,-76.478,170.678,32.650,156.137
C01216=1051.022,28.378,-76.462,170.677,32.648,156.137
C01217=1051.015,28.129,-76.446,170.675,32.646,156.137
C01218=1051.009,27.879,-76.430,170.673,32.644,156.136
C01219=1051.003,27.630,-76.414,170.671,32.642,156.136
C01220=1050.997,27.381,-76.398,170.670,32.640,156.136
C01221=1050.991,27.132,-76.382,170.668,32.638,156.135
C01222=1050.985,26.881,-76.366,170.666,32.636,156.135
C01223=1050.978,26.632,-76.350,170.665,32.634,156.135
C01224=1050.972,26.383,-76.334,170.663,32.633,156.135
C01225=1050.965,26.134,-76.318,170.661,32.631,156.134
C01226=1050.959,25.884,-76.302,170.660,32.629,156.134
C01227=1050.953,25.635,-76.286,170.658,32.627,156.134
C01228=1050.947,25.385,-76.271,170.656,32.625,156.133
C01229=1050.941,25.136,-76.255,170.654,32.623,156.133
C01230=1050.934,24.887,-76.239,170.653,32.621,156.133
C01231=1050.928,24.638,-76.223,170.652,32.619,156.132
C01232=1050.921,24.387,-76.207,170.650,32.617,156.132
C01233=1050.915,24.138,-76.191,170.649,32.615,156.132
C01234=1050.909,23.888,-76.175,170.647,32.613,156.132
C01235=1050.903,23.639,-76.159,170.645,32.611,156.131
C01236=1050.897,23.389,-76.144,170.643,32.609,156.131
C01237=1050.890,23.140,-76.128,170.642,32.607,156.131
C01238=1050.884,22.891,-76.112,170.640,32.605,156.130
C01239=1050.878,22.641,-76.097,170.638,32.603,156.130
C01240=1050.872,22.392,-76.081,170.637,32.601,156.130
C01241=1050.865,22.143,-76.065,170.635,32.599,156.130
C01242=1050.859,21.894,-76.049,170.633,32.597,156.129
C01243=1050.854,21.644,-76.033,170.631,32.596,156.129
C01244=1050.847,21.395,-76.017,170.630,32.594,156.129
C01245=1050.841,21.145,-76.001,170.628,32.592,156.128
C01246=1050.835,20.896,-75.986,170.626,32.590,156.128
C01247=1050.829,20.646,-75.970,170.625,32.588,156.128
C01248=1050.822,20.397,-75.955,170.623,32.586,156.127
C01249=1050.817,20.147,-75.939,170.621,32.584,156.127
C01250=1050.810,19.898,-75.923,170.619,32.582,156.127
C01251=1050.804,19.648,-75.908,170.618,32.580,156.127
C01252=1050.798,19.399,-75.892,170.616,32.578,156.126
C01253=1050.792,19.149,-75.876,170.614,32.576,156.126
C01254=1050.785,18.900,-75.861,170.613,32.574,156.126
C01255=1050.778,18.651,-75.845,170.612,32.572,156.125
C01256=1050.773,18.401,-75.829,170.610,32.570,156.125
C01257=1050.766,18.152,-75.814,170.608,32.569,156.125
C01258=1050.761,17.902,-75.798,170.607,32.567,156.125
C01259=1050.754,17.653,-75.783,170.605,32.565,156.124
C01260=1050.747,17.404,-75.768,170.603,32.562,156.124
C01261=1050.741,17.154,-75.751,170.601,32.560,156.124
C01262=1050.735,16.905,-75.736,170.600,32.558,156.123
C01263=1050.729,16.655,-75.720,170.598,32.557,156.123
C01264=1050.723,16.406,-75.705,170.596,32.555,156.123
C01265=1050.716,16.157,-75.690,170.595,32.553,156.123
C01266=1050.710,15.907,-75.674,170.593,32.551,156.122
C01267=1050.704,15.658,-75.658,170.591,32.549,156.122
C01268=1050.698,15.408,-75.643,170.589,32.547,156.122
C01269=1050.691,15.159,-75.627,170.588,32.546,156.122
C01270=1050.685,14.909,-75.612,170.586,32.543,156.121
C01271=1050.679,14.660,-75.596,170.584,32.541,156.121
C01272=1050.673,14.410,-75.581,170.582,32.539,156.121
C01273=1050.666,14.160,-75.566,170.581,32.537,156.120
C01274=1050.660,13.911,-75.550,170.579,32.536,156.120
C01275=1050.653,13.626,-75.533,170.577,32.534,156.120
C01276=1050.646,13.342,-75.516,170.576,32.531,156.119
C01277=1050.638,13.057,-75.498,170.574,32.529,156.119
C01278=1050.631,12.772,-75.481,170.572,32.527,156.119
C01279=1050.625,12.523,-75.466,170.570,32.526,156.119
C01280=1050.619,12.273,-75.450,170.568,32.524,156.118
C01281=1050.613,12.024,-75.435,170.567,32.522,156.118
C01282=1050.606,11.774,-75.420,170.565,32.520,156.118
C01283=1050.599,11.525,-75.404,170.563,32.518,156.118
C01284=1050.593,11.275,-75.389,170.561,32.516,156.117
C01285=1050.587,11.026,-75.374,170.560,32.514,156.117
C01286=1050.580,10.777,-75.359,170.558,32.513,156.117
C01287=1050.575,10.527,-75.343,170.556,32.511,156.117
C01288=1050.569,10.278,-75.328,170.554,32.509,156.116
C01289=1050.562,10.029,-75.313,170.552,32.507,156.116
C01290=1050.556,9.779,-75.298,170.551,32.505,156.116
C01291=1050.549,9.529,-75.283,170.549,32.503,156.115
C01292=1050.543,9.280,-75.268,170.547,32.502,156.115
C01293=1050.536,9.031,-75.252,170.545,32.500,156.115
C01294=1050.530,8.781,-75.237,170.544,32.498,156.115
C01295=1050.524,8.531,-75.222,170.542,32.496,156.114
C01296=1050.518,8.282,-75.207,170.541,32.494,156.114
C01297=1050.512,8.033,-75.192,170.539,32.492,156.114
C01298=1050.505,7.783,-75.177,170.538,32.490,156.114
C01299=1050.499,7.534,-75.162,170.536,32.489,156.113
C01300=1050.492,7.284,-75.147,170.534,32.487,156.113
C01301=1050.486,7.035,-75.132,170.532,32.484,156.113
C01302=1050.480,6.785,-75.117,170.530,32.483,156.113
C01303=1050.475,6.536,-75.102,170.529,32.481,156.112
C01304=1050.468,6.287,-75.086,170.527,32.479,156.112
C01305=1050.462,6.037,-75.071,170.525,32.478,156.112
C01306=1050.455,5.787,-75.056,170.523,32.475,156.111
C01307=1050.449,5.538,-75.041,170.522,32.474,156.111
C01308=1050.443,5.289,-75.027,170.520,32.471,156.111
C01309=1050.437,5.039,-75.012,170.518,32.470,156.111
C01310=1050.430,4.789,-74.997,170.516,32.468,156.110
C01311=1050.424,4.540,-74.981,170.514,32.466,156.110
C01312=1050.417,4.291,-74.966,170.513,32.465,156.110
C01313=1050.412,4.041,-74.951,170.511,32.462,156.110
C01314=1050.406,3.792,-74.936,170.509,32.460,156.109
C01315=1050.399,3.542,-74.921,170.507,32.459,156.109
C01316=1050.393,3.292,-74.906,170.507,32.457,156.109
C01317=1050.387,3.043,-74.891,170.505,32.455,156.109
C01318=1050.381,2.794,-74.876,170.503,32.453,156.108
C01319=1050.374,2.544,-74.862,170.501,32.451,156.108
C01320=1050.368,2.294,-74.847,170.499,32.449,156.108
C01321=1050.362,2.046,-74.832,170.498,32.447,156.107
C01322=1050.356,1.796,-74.817,170.496,32.446,156.107
C01323=1050.349,1.546,-74.802,170.494,32.444,156.107
C01324=1050.343,1.297,-74.787,170.492,32.442,156.107
C01325=1050.337,1.048,-74.773,170.491,32.440,156.106
C01326=1050.331,0.798,-74.758,170.489,32.438,156.106
C01327=1050.325,0.548,-74.743,170.487,32.436,156.106
C01328=1050.319,0.298,-74.727,170.485,32.435,156.106
C01329=1050.313,0.049,-74.713,170.483,32.433,156.105
C01330=1050.307,-0.200,-74.698,170.482,32.431,156.105
C01331=1050.300,-0.450,-74.683,170.480,32.429,156.105
C01332=1050.295,-0.699,-74.668,170.478,32.427,156.105
C01333=1050.288,-0.949,-74.653,170.476,32.425,156.104
C01334=1050.282,-1.198,-74.638,170.475,32.424,156.104
C01335=1050.276,-1.447,-74.624,170.474,32.422,156.104
C01336=1050.270,-1.697,-74.609,170.472,32.420,156.104
C01337=1050.263,-1.947,-74.594,170.470,32.418,156.103
C01338=1050.258,-2.196,-74.580,170.468,32.416,156.103
C01339=1050.250,-2.479,-74.563,170.466,32.414,156.103
C01340=1050.244,-2.761,-74.546,170.464,32.412,156.102
C01341=1050.237,-3.045,-74.530,170.462,32.410,156.102
C01342=1050.229,-3.327,-74.513,170.460,32.408,156.102
C01343=1050.223,-3.576,-74.498,170.458,32.406,156.102
C01344=1050.217,-3.826,-74.483,170.456,32.404,156.101
C01345=1050.211,-4.076,-74.469,170.455,32.402,156.101
C01346=1050.204,-4.325,-74.455,170.453,32.401,156.101
C01347=1050.198,-4.575,-74.440,170.451,32.399,156.101
C01348=1050.192,-4.824,-74.425,170.449,32.397,156.100
C01349=1050.186,-5.074,-74.411,170.447,32.395,156.100
C01350=1050.179,-5.323,-74.397,170.445,32.394,156.100
C01351=1050.173,-5.573,-74.382,170.444,32.392,156.100
C01352=1050.167,-5.822,-74.367,170.443,32.391,156.099
C01353=1050.161,-6.072,-74.353,170.441,32.388,156.099
C01354=1050.154,-6.321,-74.339,170.439,32.387,156.099
C01355=1050.148,-6.570,-74.324,170.437,32.385,156.099
C01356=1050.142,-6.820,-74.309,170.435,32.383,156.099
C01357=1050.135,-7.070,-74.295,170.434,32.381,156.098
C01358=1050.129,-7.319,-74.281,170.432,32.380,156.098
C01359=1050.123,-7.569,-74.266,170.430,32.378,156.098
C01360=1050.116,-7.819,-74.252,170.428,32.376,156.098
C01361=1050.110,-8.068,-74.238,170.426,32.374,156.097
C01362=1050.104,-8.317,-74.223,170.424,32.373,156.097
C01363=1050.098,-8.567,-74.209,170.423,32.371,156.097
C01364=1050.092,-8.816,-74.194,170.421,32.370,156.097
C01365=1050.085,-9.066,-74.180,170.419,32.367,156.096
C01366=1050.079,-9.315,-74.166,170.417,32.366,156.096
C01367=1050.073,-9.565,-74.151,170.415,32.364,156.096
C01368=1050.066,-9.814,-74.137,170.413,32.362,156.096
C01369=1050.060,-10.064,-74.123,170.412,32.360,156.095
C01370=1050.054,-10.314,-74.108,170.411,32.359,156.095
C01371=1050.048,-10.563,-74.094,170.409,32.358,156.095
C01372=1050.041,-10.812,-74.080,170.407,32.355,156.095
C01373=1050.035,-11.061,-74.065,170.405,32.354,156.094
C01374=1050.029,-11.312,-74.051,170.403,32.352,156.094
C01375=1050.023,-11.560,-74.037,170.401,32.350,156.094
C01376=1050.017,-11.811,-74.023,170.400,32.349,156.094
C01377=1050.010,-12.060,-74.008,170.398,32.347,156.094
C01378=1050.004,-12.310,-73.994,170.396,32.345,156.093
C01379=1049.998,-12.559,-73.979,170.394,32.344,156.093
C01380=1049.992,-12.809,-73.965,170.392,32.341,156.093
C01381=1049.985,-13.058,-73.951,170.390,32.340,156.093
C01382=1049.980,-13.308,-73.937,170.388,32.338,156.092
C01383=1049.973,-13.557,-73.922,170.387,32.337,156.092
C01384=1049.967,-13.807,-73.909,170.385,32.334,156.092
C01385=1049.961,-14.056,-73.894,170.383,32.333,156.092
C01386=1049.955,-14.306,-73.880,170.382,32.332,156.091
C01387=1049.948,-14.555,-73.866,170.380,32.329,156.091
C01388=1049.943,-14.805,-73.852,170.378,32.328,156.091
C01389=1049.936,-15.054,-73.837,170.376,32.326,156.091
C01390=1049.930,-15.304,-73.824,170.375,32.325,156.090
C01391=1049.924,-15.553,-73.809,170.373,32.322,156.090
C01392=1049.917,-15.803,-73.796,170.371,32.321,156.090
C01393=1049.911,-16.053,-73.782,170.369,32.320,156.090
C01394=1049.905,-16.302,-73.767,170.367,32.318,156.090
C01395=1049.898,-16.552,-73.754,170.365,32.316,156.089
C01396=1049.892,-16.801,-73.740,170.363,32.315,156.089
C01397=1049.885,-17.050,-73.726,170.361,32.313,156.089
C01398=1049.880,-17.300,-73.712,170.359,32.311,156.089
C01399=1049.873,-17.549,-73.697,170.358,32.310,156.089
C01400=1049.867,-17.799,-73.683,170.356,32.308,156.088
C01401=1049.860,-18.049,-73.670,170.354,32.306,156.088
C01402=1049.854,-18.298,-73.656,170.352,32.305,156.088
C01403=1049.847,-18.580,-73.640,170.351,32.303,156.088
C01404=1049.840,-18.861,-73.625,170.349,32.301,156.087
C01405=1049.833,-19.142,-73.609,170.346,32.299,156.087
C01406=1049.826,-19.423,-73.593,170.344,32.297,156.087
C01407=1049.819,-19.672,-73.579,170.342,32.295,156.087
C01408=1049.813,-19.922,-73.565,170.341,32.294,156.086
C01409=1049.807,-20.171,-73.552,170.339,32.293,156.086
C01410=1049.801,-20.422,-73.538,170.337,32.290,156.086
C01411=1049.795,-20.670,-73.524,170.335,32.289,156.086
C01412=1049.788,-20.920,-73.510,170.333,32.288,156.086
C01413=1049.782,-21.170,-73.496,170.331,32.286,156.085
C01414=1049.776,-21.419,-73.483,170.329,32.284,156.085
C01415=1049.770,-21.669,-73.468,170.327,32.282,156.085
C01416=1049.763,-21.918,-73.455,170.325,32.281,156.085
C01417=1049.757,-22.168,-73.441,170.323,32.279,156.085
C01418=1049.751,-22.418,-73.427,170.322,32.278,156.084
C01419=1049.745,-22.667,-73.414,170.321,32.276,156.084
C01420=1049.739,-22.917,-73.400,170.319,32.275,156.084
C01421=1049.732,-23.166,-73.386,170.317,32.273,156.084
C01422=1049.726,-23.416,-73.372,170.315,32.271,156.084
C01423=1049.720,-23.665,-73.358,170.313,32.270,156.083
C01424=1049.714,-23.915,-73.345,170.311,32.268,156.083
C01425=1049.707,-24.165,-73.331,170.309,32.266,156.083
C01426=1049.702,-24.414,-73.317,170.307,32.265,156.083
C01427=1049.695,-24.663,-73.303,170.305,32.263,156.083
C01428=1049.689,-24.913,-73.289,170.303,32.261,156.082
C01429=1049.683,-25.162,-73.276,170.302,32.260,156.082
C01430=1049.677,-25.412,-73.263,170.300,32.258,156.082
C01431=1049.670,-25.662,-73.248,170.298,32.257,156.082
C01432=1049.664,-25.911,-73.235,170.296,32.255,156.081
C01433=1049.658,-26.160,-73.222,170.294,32.253,156.081
C01434=1049.652,-26.411,-73.208,170.292,32.252,156.081
C01435=1049.646,-26.660,-73.194,170.291,32.250,156.081
C01436=1049.639,-26.909,-73.181,170.289,32.248,156.081
C01437=1049.633,-27.160,-73.167,170.287,32.247,156.080
C01438=1049.627,-27.409,-73.153,170.285,32.245,156.080
C01439=1049.620,-27.659,-73.140,170.283,32.244,156.080
C01440=1049.614,-27.908,-73.127,170.281,32.242,156.080
C01441=1049.608,-28.157,-73.113,170.279,32.241,156.080
C01442=1049.601,-28.407,-73.100,170.277,32.239,156.079
C01443=1049.595,-28.657,-73.086,170.276,32.238,156.079
C01444=1049.589,-28.906,-73.073,170.274,32.236,156.079
C01445=1049.583,-29.156,-73.059,170.272,32.234,156.079
C01446=1049.576,-29.405,-73.046,170.270,32.233,156.079
C01447=1049.570,-29.655,-73.032,170.268,32.231,156.078
C01448=1049.564,-29.904,-73.019,170.266,32.230,156.078
C01449=1049.557,-30.154,-73.005,170.264,32.229,156.078
C01450=1049.551,-30.403,-72.992,170.263,32.227,156.078
C01451=1049.545,-30.652,-72.979,170.261,32.226,156.078
C01452=1049.538,-30.902,-72.965,170.259,32.224,156.078
C01453=1049.533,-31.153,-72.952,170.257,32.223,156.077
C01454=1049.527,-31.402,-72.939,170.255,32.221,156.077
C01455=1049.520,-31.651,-72.926,170.253,32.219,156.077
C01456=1049.514,-31.901,-72.912,170.251,32.218,156.077
C01457=1049.507,-32.150,-72.899,170.249,32.216,156.077
C01458=1049.501,-32.400,-72.885,170.247,32.215,156.076
C01459=1049.494,-32.649,-72.872,170.245,32.213,156.076
C01460=1049.488,-32.899,-72.859,170.243,32.212,156.076
C01461=1049.482,-33.149,-72.846,170.241,32.210,156.076
C01462=1049.476,-33.398,-72.833,170.239,32.209,156.076
C01463=1049.470,-33.647,-72.819,170.237,32.207,156.076
C01464=1049.464,-33.897,-72.805,170.235,32.206,156.075
C01465=1049.458,-34.147,-72.793,170.233,32.204,156.075
C01466=1049.452,-34.397,-72.779,170.233,32.203,156.075
C01467=1049.444,-34.677,-72.765,170.230,32.201,156.075
C01468=1049.437,-34.957,-72.749,170.228,32.199,156.075
C01469=1049.430,-35.238,-72.735,170.226,32.198,156.074
C01470=1049.423,-35.518,-72.719,170.224,32.196,156.074
C01471=1049.418,-35.768,-72.707,170.222,32.194,156.074
C01472=1049.411,-36.017,-72.693,170.220,32.193,156.074
C01473=1049.405,-36.266,-72.680,170.218,32.191,156.074
C01474=1049.399,-36.517,-72.667,170.216,32.190,156.073
C01475=1049.392,-36.766,-72.654,170.214,32.188,156.073
C01476=1049.386,-37.015,-72.641,170.212,32.187,156.073
C01477=1049.380,-37.265,-72.627,170.210,32.185,156.073
C01478=1049.374,-37.515,-72.615,170.208,32.184,156.073
C01479=1049.368,-37.764,-72.602,170.206,32.182,156.073
C01480=1049.361,-38.014,-72.588,170.204,32.181,156.072
C01481=1049.355,-38.264,-72.575,170.203,32.180,156.072
C01482=1049.349,-38.513,-72.562,170.201,32.178,156.072
C01483=1049.343,-38.762,-72.549,170.199,32.177,156.072
C01484=1049.337,-39.012,-72.536,170.197,32.175,156.072
C01485=1049.331,-39.261,-72.523,170.195,32.174,156.071
C01486=1049.324,-39.512,-72.510,170.193,32.172,156.071
C01487=1049.318,-39.761,-72.497,170.191,32.171,156.071
C01488=1049.311,-40.010,-72.484,170.189,32.170,156.071
C01489=1049.305,-40.260,-72.472,170.187,32.168,156.071
C01490=1049.299,-40.509,-72.458,170.185,32.167,156.071
C01491=1049.293,-40.759,-72.446,170.183,32.165,156.071
C01492=1049.287,-41.008,-72.433,170.181,32.164,156.070
C01493=1049.280,-41.259,-72.420,170.179,32.162,156.070
C01494=1049.273,-41.508,-72.407,170.177,32.161,156.070
C01495=1049.267,-41.758,-72.394,170.175,32.160,156.070
C01496=1049.261,-42.007,-72.381,170.174,32.159,156.070
C01497=1049.255,-42.257,-72.369,170.172,32.157,156.070
C01498=1049.249,-42.506,-72.355,170.170,32.156,156.069
C01499=1049.242,-42.756,-72.343,170.168,32.154,156.069
C01500=1049.236,-43.005,-72.330,170.166,32.153,156.069
C01501=1049.230,-43.255,-72.318,170.164,32.151,156.069
C01502=1049.223,-43.505,-72.304,170.162,32.150,156.069
C01503=1049.217,-43.755,-72.291,170.160,32.149,156.069
C01504=1049.210,-44.004,-72.279,170.158,32.147,156.068
C01505=1049.205,-44.254,-72.266,170.156,32.146,156.068
C01506=1049.198,-44.503,-72.253,170.154,32.144,156.068
C01507=1049.192,-44.753,-72.240,170.152,32.143,156.068
C01508=1049.187,-45.003,-72.228,170.150,32.142,156.068
C01509=1049.180,-45.252,-72.215,170.148,32.141,156.068
C01510=1049.174,-45.502,-72.203,170.146,32.139,156.068
C01511=1049.167,-45.751,-72.189,170.145,32.138,156.067
C01512=1049.162,-46.001,-72.177,170.143,32.136,156.067
C01513=1049.155,-46.250,-72.165,170.141,32.135,156.067
C01514=1049.149,-46.500,-72.152,170.139,32.134,156.067
C01515=1049.143,-46.749,-72.139,170.137,32.132,156.067
C01516=1049.137,-46.999,-72.126,170.135,32.131,156.067
C01517=1049.131,-47.249,-72.113,170.133,32.129,156.066
C01518=1049.124,-47.498,-72.101,170.131,32.128,156.066
C01519=1049.118,-47.747,-72.088,170.128,32.127,156.066
C01520=1049.112,-47.997,-72.075,170.126,32.125,156.066
C01521=1049.106,-48.247,-72.063,170.124,32.124,156.066
C01522=1049.099,-48.497,-72.051,170.122,32.122,156.066
C01523=1049.093,-48.746,-72.038,170.120,32.121,156.066
C01524=1049.087,-48.996,-72.025,170.118,32.120,156.065
C01525=1049.081,-49.246,-72.012,170.116,32.119,156.065
C01526=1049.074,-49.495,-72.000,170.115,32.117,156.065
C01527=1049.068,-49.745,-71.987,170.113,32.116,156.065
C01528=1049.063,-49.995,-71.975,170.111,32.115,156.065
C01529=1049.057,-50.244,-71.962,170.109,32.113,156.065
C01530=1049.050,-50.493,-71.949,170.107,32.112,156.065
C01531=1049.043,-50.775,-71.936,170.105,32.110,156.064
C01532=1049.036,-51.056,-71.922,170.102,32.109,156.064
C01533=1049.028,-51.337,-71.908,170.100,32.108,156.064
C01534=1049.022,-51.617,-71.894,170.098,32.106,156.064
C01535=1049.015,-51.867,-71.882,170.096,32.105,156.064
C01536=1049.009,-52.117,-71.870,170.094,32.104,156.064
C01537=1049.002,-52.366,-71.857,170.092,32.103,156.064
C01538=1048.995,-52.615,-71.845,170.089,32.102,156.064
C01539=1048.990,-52.865,-71.832,170.087,32.100,156.063
C01540=1048.983,-53.115,-71.820,170.086,32.099,156.063
C01541=1048.977,-53.365,-71.808,170.084,32.098,156.063
C01542=1048.970,-53.614,-71.796,170.082,32.097,156.063
C01543=1048.964,-53.864,-71.783,170.080,32.095,156.063
C01544=1048.958,-54.114,-71.771,170.078,32.095,156.063
C01545=1048.951,-54.363,-71.759,170.076,32.093,156.063
C01546=1048.945,-54.612,-71.746,170.074,32.092,156.063
C01547=1048.938,-54.862,-71.734,170.072,32.091,156.062
C01548=1048.932,-55.112,-71.722,170.070,32.090,156.062
C01549=1048.926,-55.361,-71.710,170.068,32.088,156.062
C01550=1048.919,-55.611,-71.698,170.066,32.088,156.062
C01551=1048.913,-55.861,-71.685,170.063,32.086,156.062
C01552=1048.907,-56.110,-71.673,170.061,32.085,156.062
C01553=1048.901,-56.360,-71.661,170.059,32.084,156.062
C01554=1048.895,-56.609,-71.649,170.057,32.083,156.062
C01555=1048.888,-56.859,-71.637,170.055,32.081,156.062
C01556=1048.882,-57.109,-71.625,170.054,32.080,156.061
C01557=1048.875,-57.358,-71.613,170.052,32.079,156.061
C01558=1048.869,-57.608,-71.601,170.050,32.078,156.061
C01559=1048.863,-57.858,-71.588,170.048,32.076,156.061
C01560=1048.856,-58.107,-71.576,170.046,32.076,156.061
C01561=1048.850,-58.357,-71.564,170.044,32.074,156.061
C01562=1048.845,-58.607,-71.553,170.041,32.073,156.061
C01563=1048.838,-58.856,-71.541,170.039,32.072,156.061
C01564=1048.832,-59.106,-71.528,170.037,32.071,156.061
C01565=1048.825,-59.356,-71.516,170.035,32.069,156.060
C01566=1048.819,-59.605,-71.504,170.033,32.068,156.060
C01567=1048.813,-59.855,-71.492,170.031,32.067,156.060
C01568=1048.806,-60.105,-71.480,170.029,32.066,156.060
C01569=1048.800,-60.354,-71.468,170.027,32.065,156.060
C01570=1048.794,-60.603,-71.456,170.025,32.064,156.060
C01571=1048.787,-60.853,-71.444,170.024,32.063,156.060
C01572=1048.781,-61.103,-71.432,170.021,32.061,156.060
C01573=1048.775,-61.353,-71.420,170.019,32.060,156.060
C01574=1048.769,-61.602,-71.408,170.017,32.059,156.059
C01575=1048.763,-61.852,-71.396,170.015,32.058,156.059
C01576=1048.757,-62.101,-71.384,170.013,32.057,156.059
C01577=1048.750,-62.351,-71.372,170.011,32.056,156.059
C01578=1048.744,-62.601,-71.361,170.009,32.055,156.059
C01579=1048.738,-62.850,-71.348,170.007,32.053,156.059
C01580=1048.732,-63.100,-71.336,170.005,32.052,156.059
C01581=1048.725,-63.350,-71.324,170.003,32.051,156.059
C01582=1048.719,-63.599,-71.312,170.000,32.050,156.059
C01583=1048.713,-63.849,-71.301,169.998,32.049,156.059
C01584=1048.707,-64.098,-71.289,169.996,32.048,156.058
C01585=1048.701,-64.348,-71.277,169.994,32.047,156.058
C01586=1048.694,-64.598,-71.265,169.993,32.045,156.058
C01587=1048.688,-64.847,-71.254,169.991,32.044,156.058
C01588=1048.682,-65.097,-71.242,169.989,32.044,156.058
C01589=1048.676,-65.347,-71.229,169.987,32.042,156.058
C01590=1048.670,-65.596,-71.218,169.985,32.041,156.058
C01591=1048.664,-65.846,-71.206,169.982,32.040,156.058
C01592=1048.658,-66.096,-71.194,169.980,32.039,156.058
C01593=1048.651,-66.345,-71.182,169.978,32.038,156.058
C01594=1048.645,-66.595,-71.171,169.976,32.036,156.057
C01595=1048.636,-66.970,-71.153,169.973,32.035,156.057
C01596=1048.626,-67.345,-71.135,169.970,32.033,156.057
C01597=1048.618,-67.720,-71.117,169.967,32.032,156.057
C01598=1048.608,-68.095,-71.100,169.963,32.030,156.057
C01599=1048.602,-68.345,-71.088,169.962,32.029,156.057
C01600=1048.596,-68.594,-71.077,169.960,32.028,156.057
C01601=1048.589,-68.844,-71.065,169.958,32.027,156.057
C01602=1048.584,-69.094,-71.053,169.956,32.026,156.056
C01603=1048.578,-69.343,-71.041,169.954,32.025,156.056
C01604=1048.571,-69.593,-71.029,169.952,32.023,156.056
C01605=1048.566,-69.842,-71.018,169.949,32.022,156.056
C01606=1048.560,-70.092,-71.006,169.947,32.021,156.056
C01607=1048.553,-70.342,-70.995,169.945,32.020,156.056
C01608=1048.547,-70.591,-70.983,169.943,32.019,156.056
C01609=1048.542,-70.842,-70.971,169.941,32.018,156.056
C01610=1048.535,-71.090,-70.960,169.939,32.017,156.056
C01611=1048.529,-71.341,-70.948,169.937,32.016,156.056
C01612=1048.523,-71.590,-70.936,169.935,32.015,156.056
C01613=1048.517,-71.840,-70.926,169.932,32.014,156.056
C01614=1048.511,-72.090,-70.913,169.931,32.013,156.055
C01615=1048.505,-72.339,-70.902,169.929,32.012,156.055
C01616=1048.498,-72.589,-70.890,169.927,32.011,156.055
C01617=1048.493,-72.838,-70.879,169.925,32.009,156.055
C01618=1048.487,-73.088,-70.867,169.923,32.008,156.055
C01619=1048.480,-73.338,-70.856,169.921,32.008,156.055
C01620=1048.474,-73.587,-70.844,169.918,32.007,156.055
C01621=1048.468,-73.837,-70.833,169.916,32.005,156.055
C01622=1048.462,-74.086,-70.821,169.914,32.004,156.055
C01623=1048.456,-74.336,-70.810,169.912,32.003,156.055
C01624=1048.450,-74.586,-70.799,169.910,32.002,156.055
C01625=1048.443,-74.835,-70.787,169.908,32.002,156.055
C01626=1048.437,-75.086,-70.776,169.906,32.001,156.054
C01627=1048.431,-75.335,-70.765,169.903,32.000,156.054
C01628=1048.425,-75.585,-70.753,169.901,31.999,156.054
C01629=1048.419,-75.834,-70.742,169.900,31.998,156.054
C01630=1048.412,-76.084,-70.730,169.898,31.997,156.054
C01631=1048.402,-76.490,-70.712,169.894,31.995,156.054
C01632=1048.393,-76.897,-70.693,169.891,31.994,156.054
C01633=1048.383,-77.304,-70.675,169.887,31.992,156.054
C01634=1048.373,-77.710,-70.657,169.884,31.991,156.054
C01635=1048.366,-77.960,-70.645,169.882,31.990,156.054
C01636=1048.360,-78.209,-70.635,169.879,31.989,156.054
C01637=1048.353,-78.459,-70.623,169.877,31.988,156.054
C01638=1048.348,-78.709,-70.613,169.875,31.987,156.054
C01639=1048.341,-78.958,-70.601,169.873,31.987,156.054
C01640=1048.335,-79.208,-70.590,169.871,31.986,156.054
C01641=1048.329,-79.458,-70.578,169.869,31.985,156.053
C01642=1048.323,-79.707,-70.568,169.867,31.984,156.053
C01643=1048.317,-79.957,-70.556,169.865,31.983,156.053
C01644=1048.311,-80.206,-70.545,169.863,31.982,156.053
C01645=1048.304,-80.456,-70.534,169.861,31.981,156.053
C01646=1048.298,-80.706,-70.523,169.859,31.980,156.053
C01647=1048.292,-80.956,-70.512,169.856,31.979,156.053
C01648=1048.286,-81.205,-70.501,169.854,31.978,156.053
C01649=1048.279,-81.455,-70.490,169.852,31.978,156.053
C01650=1048.273,-81.704,-70.479,169.850,31.977,156.053
C01651=1048.266,-81.954,-70.468,169.848,31.976,156.053
C01652=1048.261,-82.204,-70.457,169.845,31.975,156.053
C01653=1048.254,-82.454,-70.446,169.843,31.975,156.053
C01654=1048.248,-82.703,-70.435,169.841,31.974,156.053
C01655=1048.241,-82.987,-70.423,169.838,31.973,156.053
C01656=1048.234,-83.273,-70.410,169.836,31.972,156.053
C01657=1048.226,-83.557,-70.398,169.834,31.971,156.053
C01658=1048.219,-83.841,-70.385,169.832,31.971,156.053
C01659=1048.212,-84.090,-70.374,169.830,31.970,156.053
C01660=1048.207,-84.340,-70.363,169.828,31.969,156.053
C01661=1048.201,-84.589,-70.353,169.825,31.968,156.053
C01662=1048.194,-84.839,-70.342,169.823,31.967,156.053
C01663=1048.188,-85.089,-70.331,169.821,31.967,156.053
C01664=1048.182,-85.339,-70.320,169.819,31.966,156.053
C01665=1048.176,-85.589,-70.309,169.816,31.965,156.053
C01666=1048.169,-85.838,-70.298,169.814,31.964,156.053
C01667=1048.163,-86.088,-70.287,169.812,31.963,156.052
C01668=1048.157,-86.337,-70.276,169.810,31.963,156.052
C01669=1048.150,-86.587,-70.266,169.808,31.962,156.052
C01670=1048.145,-86.837,-70.255,169.805,31.961,156.052
C01671=1048.138,-87.087,-70.244,169.803,31.960,156.052
C01672=1048.132,-87.336,-70.233,169.801,31.960,156.052
C01673=1048.126,-87.586,-70.223,169.799,31.959,156.052
C01674=1048.120,-87.836,-70.211,169.798,31.958,156.052
C01675=1048.113,-88.085,-70.201,169.795,31.957,156.052
C01676=1048.108,-88.335,-70.191,169.793,31.957,156.052
C01677=1048.101,-88.585,-70.180,169.791,31.956,156.052
C01678=1048.095,-88.834,-70.169,169.789,31.955,156.052
C01679=1048.089,-89.084,-70.158,169.786,31.955,156.052
C01680=1048.083,-89.334,-70.147,169.784,31.954,156.052
C01681=1048.076,-89.583,-70.137,169.782,31.953,156.052
C01682=1048.071,-89.833,-70.126,169.780,31.952,156.052
C01683=1048.064,-90.083,-70.115,169.778,31.952,156.052
C01684=1048.058,-90.333,-70.105,169.775,31.951,156.052
C01685=1048.052,-90.582,-70.094,169.773,31.950,156.052
C01686=1048.045,-90.832,-70.084,169.771,31.950,156.052
C01687=1048.040,-91.082,-70.073,169.769,31.949,156.052
C01688=1048.034,-91.331,-70.062,169.767,31.948,156.052
C01689=1048.027,-91.581,-70.051,169.764,31.948,156.052
C01690=1048.021,-91.831,-70.041,169.763,31.947,156.052
C01691=1048.015,-92.080,-70.031,169.761,31.946,156.052
C01692=1048.009,-92.330,-70.020,169.759,31.946,156.052
C01693=1048.003,-92.580,-70.009,169.756,31.945,156.052
C01694=1047.996,-92.829,-69.998,169.754,31.944,156.052
C01695=1047.991,-93.079,-69.988,169.752,31.944,156.052
C01696=1047.985,-93.329,-69.977,169.750,31.943,156.052
C01697=1047.978,-93.579,-69.967,169.747,31.942,156.052
C01698=1047.972,-93.828,-69.956,169.745,31.941,156.052
C01699=1047.966,-94.078,-69.946,169.743,31.941,156.052
C01700=1047.960,-94.327,-69.935,169.741,31.940,156.052
C01701=1047.954,-94.578,-69.924,169.739,31.939,156.052
C01702=1047.948,-94.827,-69.915,169.736,31.938,156.052
C01703=1047.942,-95.077,-69.904,169.734,31.938,156.052
C01704=1047.936,-95.326,-69.893,169.732,31.937,156.052
C01705=1047.930,-95.576,-69.883,169.730,31.937,156.052
C01706=1047.924,-95.826,-69.872,169.727,31.936,156.052
C01707=1047.917,-96.076,-69.862,169.726,31.935,156.052
C01708=1047.912,-96.325,-69.851,169.724,31.935,156.052
C01709=1047.906,-96.575,-69.841,169.722,31.934,156.052
C01710=1047.900,-96.824,-69.830,169.719,31.934,156.052
C01711=1047.893,-97.075,-69.821,169.717,31.933,156.052
C01712=1047.887,-97.324,-69.810,169.715,31.932,156.052
C01713=1047.882,-97.574,-69.799,169.713,31.932,156.052
C01714=1047.875,-97.824,-69.789,169.711,31.931,156.052
C01715=1047.869,-98.073,-69.779,169.708,31.930,156.052
C01716=1047.863,-98.324,-69.768,169.706,31.930,156.052
C01717=1047.856,-98.573,-69.758,169.704,31.929,156.052
C01718=1047.850,-98.823,-69.749,169.701,31.929,156.052
C01719=1047.843,-99.110,-69.736,169.699,31.928,156.052
C01720=1047.836,-99.396,-69.724,169.696,31.928,156.052
C01721=1047.829,-99.682,-69.712,169.694,31.927,156.052
C01722=1047.822,-99.969,-69.702,169.691,31.926,156.052
C01723=1047.816,-100.218,-69.691,169.690,31.926,156.052
C01724=1047.810,-100.469,-69.681,169.688,31.925,156.052
C01725=1047.803,-100.718,-69.671,169.685,31.925,156.052
C01726=1047.798,-100.968,-69.660,169.683,31.925,156.052
C01727=1047.791,-101.217,-69.650,169.681,31.924,156.052
C01728=1047.785,-101.467,-69.640,169.679,31.924,156.052
C01729=1047.779,-101.717,-69.630,169.676,31.923,156.052
C01730=1047.773,-101.966,-69.620,169.674,31.922,156.052
C01731=1047.766,-102.216,-69.609,169.672,31.922,156.052
C01732=1047.761,-102.466,-69.599,169.669,31.922,156.052
C01733=1047.754,-102.716,-69.590,169.667,31.921,156.052
C01734=1047.748,-102.965,-69.579,169.665,31.921,156.052
C01735=1047.742,-103.215,-69.570,169.663,31.920,156.052
C01736=1047.736,-103.465,-69.559,169.660,31.919,156.052
C01737=1047.730,-103.714,-69.549,169.658,31.919,156.052
C01738=1047.724,-103.964,-69.540,169.656,31.919,156.052
C01739=1047.718,-104.214,-69.529,169.654,31.918,156.052
C01740=1047.712,-104.464,-69.519,169.651,31.918,156.052
C01741=1047.705,-104.714,-69.509,169.650,31.917,156.052
C01742=1047.698,-104.963,-69.499,169.648,31.917,156.053
C01743=1047.693,-105.213,-69.489,169.646,31.916,156.052
C01744=1047.687,-105.463,-69.479,169.643,31.916,156.053
C01745=1047.680,-105.712,-69.469,169.641,31.916,156.053
C01746=1047.675,-105.962,-69.459,169.639,31.915,156.053
C01747=1047.669,-106.212,-69.449,169.636,31.914,156.053
C01748=1047.662,-106.461,-69.439,169.634,31.914,156.053
C01749=1047.656,-106.711,-69.430,169.632,31.914,156.053
C01750=1047.650,-106.961,-69.420,169.630,31.914,156.053
C01751=1047.644,-107.210,-69.409,169.627,31.913,156.053
C01752=1047.638,-107.460,-69.400,169.625,31.912,156.053
C01753=1047.632,-107.710,-69.390,169.623,31.912,156.053
C01754=1047.626,-107.960,-69.380,169.621,31.912,156.053
C01755=1047.620,-108.210,-69.371,169.618,31.911,156.053
C01756=1047.613,-108.459,-69.361,169.616,31.911,156.053
C01757=1047.608,-108.709,-69.350,169.614,31.911,156.053
C01758=1047.601,-108.959,-69.341,169.611,31.911,156.053
C01759=1047.595,-109.209,-69.331,169.609,31.910,156.053
C01760=1047.589,-109.458,-69.322,169.608,31.909,156.053
C01761=1047.583,-109.708,-69.311,169.605,31.909,156.053
C01762=1047.576,-109.957,-69.302,169.603,31.909,156.053
C01763=1047.570,-110.207,-69.292,169.601,31.909,156.053
C01764=1047.564,-110.457,-69.283,169.599,31.908,156.053
C01765=1047.558,-110.707,-69.273,169.596,31.908,156.053
C01766=1047.552,-110.957,-69.264,169.594,31.908,156.054
C01767=1047.546,-111.206,-69.253,169.592,31.907,156.054
C01768=1047.540,-111.456,-69.243,169.589,31.907,156.054
C01769=1047.534,-111.706,-69.234,169.587,31.907,156.054
C01770=1047.528,-111.955,-69.224,169.585,31.907,156.054
C01771=1047.521,-112.205,-69.214,169.583,31.906,156.054
C01772=1047.515,-112.455,-69.205,169.580,31.906,156.054
C01773=1047.509,-112.705,-69.195,169.578,31.906,156.054
C01774=1047.503,-112.955,-69.186,169.576,31.905,156.054
C01775=1047.497,-113.204,-69.176,169.573,31.905,156.054
C01776=1047.490,-113.454,-69.167,169.571,31.905,156.054
C01777=1047.484,-113.704,-69.157,169.569,31.905,156.054
C01778=1047.478,-113.954,-69.147,169.567,31.904,156.054
C01779=1047.472,-114.204,-69.138,169.565,31.904,156.054
C01780=1047.466,-114.453,-69.128,169.563,31.904,156.054
C01781=1047.460,-114.703,-69.119,169.561,31.903,156.054
C01782=1047.454,-114.952,-69.110,169.558,31.903,156.055
C01783=1047.447,-115.238,-69.098,169.556,31.903,156.055
C01784=1047.440,-115.523,-69.087,169.553,31.902,156.055
C01785=1047.433,-115.809,-69.076,169.550,31.902,156.055
C01786=1047.426,-116.095,-69.066,169.548,31.902,156.055
C01787=1047.420,-116.345,-69.056,169.545,31.902,156.055
C01788=1047.414,-116.594,-69.047,169.543,31.901,156.055
C01789=1047.407,-116.844,-69.037,169.541,31.902,156.055
C01790=1047.401,-117.094,-69.028,169.539,31.901,156.055
C01791=1047.395,-117.344,-69.018,169.536,31.901,156.055
C01792=1047.390,-117.593,-69.009,169.534,31.901,156.055
C01793=1047.383,-117.843,-68.999,169.532,31.901,156.055
C01794=1047.377,-118.092,-68.990,169.529,31.900,156.055
C01795=1047.370,-118.342,-68.981,169.527,31.900,156.055
C01796=1047.364,-118.592,-68.971,169.525,31.900,156.056
C01797=1047.358,-118.842,-68.962,169.522,31.900,156.056
C01798=1047.352,-119.092,-68.953,169.521,31.900,156.056
C01799=1047.347,-119.341,-68.944,169.519,31.899,156.056
C01800=1047.340,-119.591,-68.934,169.516,31.899,156.056
C01801=1047.334,-119.841,-68.924,169.514,31.899,156.056
C01802=1047.328,-120.090,-68.915,169.512,31.899,156.056
C01803=1047.322,-120.341,-68.906,169.509,31.899,156.056
C01804=1047.315,-120.590,-68.897,169.507,31.899,156.056
C01805=1047.310,-120.839,-68.888,169.505,31.898,156.056
C01806=1047.304,-121.089,-68.878,169.503,31.899,156.057
C01807=1047.297,-121.339,-68.869,169.500,31.898,156.057
C01808=1047.291,-121.589,-68.860,169.498,31.898,156.057
C01809=1047.285,-121.839,-68.850,169.496,31.898,156.057
C01810=1047.279,-122.088,-68.842,169.493,31.898,156.057
C01811=1047.273,-122.338,-68.832,169.491,31.898,156.057
C01812=1047.267,-122.588,-68.823,169.489,31.898,156.057
C01813=1047.261,-122.838,-68.814,169.486,31.898,156.057
